C05469=1110.631,164.327,-63.571,-179.323,8.948,149.553
C05470=1110.636,164.078,-63.548,-179.324,8.945,149.553
C05471=1110.640,163.829,-63.525,-179.327,8.942,149.553
C05472=1110.644,163.580,-63.502,-179.329,8.939,149.553
C05473=1110.649,163.331,-63.479,-179.331,8.936,149.553
C05474=1110.654,163.082,-63.455,-179.334,8.932,149.552
C05475=1110.658,162.834,-63.432,-179.335,8.930,149.552
C05476=1110.663,162.585,-63.410,-179.338,8.926,149.552
C05477=1110.667,162.336,-63.387,-179.340,8.923,149.552
C05478=1110.672,162.087,-63.364,-179.342,8.920,149.552
C05479=1110.677,161.838,-63.341,-179.344,8.917,149.552
C05480=1110.681,161.588,-63.319,-179.346,8.914,149.551
C05481=1110.686,161.340,-63.296,-179.349,8.911,149.551
C05482=1110.690,161.091,-63.273,-179.351,8.907,149.551
C05483=1110.695,160.842,-63.249,-179.353,8.905,149.551
C05484=1110.699,160.593,-63.227,-179.355,8.902,149.551
C05485=1110.703,160.380,-63.208,-179.357,8.899,149.551
C05486=1110.707,160.167,-63.188,-179.359,8.896,149.551
C05487=1110.711,159.953,-63.168,-179.361,8.893,149.551
C05488=1110.715,159.739,-63.149,-179.362,8.891,149.550
C05489=1110.719,159.527,-63.129,-179.365,8.888,149.550
C05490=1110.723,159.312,-63.110,-179.366,8.885,149.550
C05491=1110.727,159.099,-63.090,-179.368,8.883,149.550
C05492=1110.731,158.886,-63.071,-179.369,8.880,149.550
C05493=1110.735,158.637,-63.048,-179.372,8.877,149.550
C05494=1110.740,158.388,-63.025,-179.374,8.873,149.550
C05495=1110.744,158.139,-63.003,-179.376,8.870,149.550
C05496=1110.750,157.890,-62.980,-179.379,8.867,149.549
C05497=1110.754,157.641,-62.958,-179.380,8.864,149.549
C05498=1110.758,157.392,-62.936,-179.382,8.861,149.549
C05499=1110.763,157.144,-62.913,-179.385,8.857,149.549
C05500=1110.767,156.895,-62.890,-179.387,8.854,149.549
C05501=1110.772,156.645,-62.867,-179.389,8.851,149.549
C05502=1110.777,156.397,-62.845,-179.391,8.847,149.548
C05503=1110.782,156.148,-62.822,-179.393,8.844,149.548
C05504=1110.786,155.899,-62.799,-179.395,8.841,149.548
C05505=1110.791,155.650,-62.778,-179.397,8.838,149.548
C05506=1110.795,155.401,-62.754,-179.399,8.834,149.548
C05507=1110.800,155.152,-62.732,-179.401,8.831,149.547
C05508=1110.805,154.903,-62.711,-179.404,8.828,149.547
C05509=1110.809,154.654,-62.687,-179.406,8.824,149.547
C05510=1110.814,154.405,-62.665,-179.408,8.821,149.547
C05511=1110.819,154.156,-62.642,-179.410,8.817,149.547
C05512=1110.823,153.907,-62.620,-179.412,8.815,149.546
C05513=1110.827,153.658,-62.598,-179.414,8.812,149.546
C05514=1110.833,153.409,-62.575,-179.416,8.808,149.546
C05515=1110.837,153.160,-62.553,-179.418,8.805,149.546
C05516=1110.841,152.911,-62.531,-179.420,8.801,149.546
C05517=1110.847,152.662,-62.508,-179.423,8.798,149.545
C05518=1110.851,152.413,-62.486,-179.425,8.794,149.545
C05519=1110.856,152.164,-62.464,-179.427,8.791,149.545
C05520=1110.860,151.916,-62.442,-179.429,8.788,149.545
C05521=1110.865,151.666,-62.419,-179.431,8.784,149.545
C05522=1110.870,151.417,-62.397,-179.433,8.781,149.544
C05523=1110.874,151.168,-62.375,-179.435,8.777,149.544
C05524=1110.878,150.920,-62.353,-179.438,8.774,149.544
C05525=1110.883,150.670,-62.330,-179.440,8.770,149.544
C05526=1110.888,150.422,-62.308,-179.442,8.767,149.543
C05527=1110.892,150.172,-62.286,-179.444,8.763,149.543
C05528=1110.897,149.924,-62.264,-179.446,8.760,149.543
C05529=1110.902,149.675,-62.241,-179.447,8.757,149.543
C05530=1110.906,149.425,-62.219,-179.449,8.753,149.543
C05531=1110.911,149.177,-62.198,-179.451,8.750,149.542
C05532=1110.915,148.927,-62.176,-179.454,8.747,149.542
C05533=1110.920,148.679,-62.154,-179.456,8.743,149.542
C05534=1110.925,148.429,-62.132,-179.458,8.740,149.542
C05535=1110.930,148.181,-62.109,-179.460,8.735,149.541
C05536=1110.934,147.932,-62.087,-179.463,8.732,149.541
C05537=1110.939,147.683,-62.065,-179.465,8.728,149.541
C05538=1110.943,147.434,-62.043,-179.466,8.724,149.540
C05539=1110.948,147.185,-62.021,-179.468,8.721,149.540
C05540=1110.952,146.936,-61.999,-179.470,8.717,149.540
C05541=1110.957,146.722,-61.981,-179.472,8.715,149.540
C05542=1110.960,146.508,-61.962,-179.474,8.711,149.539
C05543=1110.965,146.296,-61.943,-179.475,8.709,149.539
C05544=1110.968,146.082,-61.924,-179.477,8.705,149.539
C05545=1110.973,145.868,-61.905,-179.479,8.702,149.539
C05546=1110.977,145.654,-61.886,-179.481,8.699,149.539
C05547=1110.981,145.441,-61.868,-179.482,8.696,149.538
C05548=1110.985,145.227,-61.848,-179.485,8.693,149.538
C05549=1110.990,144.979,-61.827,-179.486,8.690,149.538
C05550=1110.994,144.730,-61.805,-179.488,8.686,149.537
C05551=1110.999,144.480,-61.784,-179.489,8.682,149.537
C05552=1111.004,144.232,-61.762,-179.491,8.679,149.537
C05553=1111.008,143.982,-61.740,-179.492,8.676,149.536
C05554=1111.013,143.734,-61.718,-179.494,8.672,149.536
C05555=1111.017,143.484,-61.696,-179.496,8.668,149.536
C05556=1111.022,143.236,-61.675,-179.497,8.666,149.535
C05557=1111.027,142.987,-61.653,-179.499,8.662,149.535
C05558=1111.031,142.738,-61.631,-179.501,8.658,149.535
C05559=1111.036,142.489,-61.609,-179.503,8.655,149.534
C05560=1111.041,142.239,-61.588,-179.504,8.652,149.534
C05561=1111.046,141.990,-61.566,-179.506,8.648,149.534
C05562=1111.049,141.741,-61.545,-179.507,8.645,149.533
C05563=1111.054,141.493,-61.523,-179.509,8.642,149.533
C05564=1111.059,141.244,-61.501,-179.511,8.638,149.533
C05565=1111.063,140.994,-61.480,-179.513,8.635,149.532
C05566=1111.068,140.745,-61.458,-179.515,8.631,149.532
C05567=1111.073,140.497,-61.437,-179.516,8.628,149.532
C05568=1111.077,140.247,-61.415,-179.518,8.624,149.532
C05569=1111.083,139.998,-61.394,-179.519,8.621,149.531
C05570=1111.087,139.750,-61.372,-179.521,8.618,149.531
C05571=1111.092,139.500,-61.350,-179.523,8.614,149.531
C05572=1111.097,139.251,-61.329,-179.524,8.611,149.530
C05573=1111.100,139.002,-61.307,-179.527,8.607,149.530
C05574=1111.105,138.753,-61.286,-179.529,8.604,149.530
C05575=1111.110,138.505,-61.264,-179.530,8.601,149.529
C05576=1111.115,138.255,-61.243,-179.532,8.597,149.529
C05577=1111.120,138.006,-61.221,-179.533,8.594,149.529
C05578=1111.125,137.757,-61.200,-179.535,8.591,149.528
C05579=1111.129,137.508,-61.179,-179.537,8.587,149.528
C05580=1111.133,137.259,-61.157,-179.538,8.583,149.528
C05581=1111.138,137.010,-61.136,-179.540,8.581,149.528
C05582=1111.143,136.761,-61.114,-179.542,8.577,149.527
C05583=1111.148,136.511,-61.093,-179.544,8.573,149.527
C05584=1111.152,136.263,-61.072,-179.545,8.571,149.527
C05585=1111.157,136.014,-61.050,-179.547,8.567,149.526
C05586=1111.161,135.764,-61.029,-179.549,8.563,149.526
C05587=1111.166,135.516,-61.007,-179.550,8.561,149.526
C05588=1111.171,135.267,-60.987,-179.552,8.557,149.525
C05589=1111.176,135.018,-60.965,-179.554,8.553,149.525
C05590=1111.180,134.768,-60.944,-179.555,8.550,149.525
C05591=1111.185,134.519,-60.922,-179.557,8.547,149.525
C05592=1111.189,134.271,-60.902,-179.560,8.544,149.524
C05593=1111.194,134.022,-60.880,-179.561,8.540,149.524
C05594=1111.199,133.772,-60.859,-179.563,8.537,149.524
C05595=1111.204,133.523,-60.837,-179.565,8.533,149.523
C05596=1111.208,133.274,-60.817,-179.566,8.530,149.523
C05597=1111.213,133.061,-60.798,-179.568,8.527,149.523
C05598=1111.217,132.846,-60.780,-179.569,8.524,149.523
C05599=1111.220,132.633,-60.762,-179.571,8.521,149.522
C05600=1111.224,132.420,-60.744,-179.572,8.519,149.522
C05601=1111.228,132.206,-60.726,-179.574,8.516,149.522
C05602=1111.233,131.992,-60.707,-179.575,8.513,149.522
C05603=1111.237,131.779,-60.689,-179.577,8.510,149.521
C05604=1111.241,131.565,-60.672,-179.578,8.507,149.521
C05605=1111.245,131.316,-60.650,-179.579,8.504,149.521
C05606=1111.250,131.067,-60.630,-179.582,8.500,149.521
C05607=1111.255,130.818,-60.609,-179.584,8.497,149.520
C05608=1111.260,130.569,-60.587,-179.585,8.494,149.520
C05609=1111.264,130.320,-60.567,-179.587,8.490,149.520
C05610=1111.269,130.071,-60.546,-179.589,8.487,149.519
C05611=1111.273,129.822,-60.524,-179.590,8.484,149.519
C05612=1111.278,129.572,-60.503,-179.592,8.481,149.519
C05613=1111.283,129.323,-60.482,-179.594,8.477,149.518
C05614=1111.288,129.074,-60.462,-179.595,8.474,149.518
C05615=1111.292,128.826,-60.440,-179.597,8.471,149.518
C05616=1111.297,128.577,-60.420,-179.599,8.467,149.518
C05617=1111.302,128.327,-60.399,-179.600,8.464,149.517
C05618=1111.306,128.078,-60.378,-179.603,8.461,149.517
C05619=1111.311,127.828,-60.357,-179.605,8.457,149.517
C05620=1111.315,127.580,-60.336,-179.606,8.454,149.517
C05621=1111.320,127.331,-60.315,-179.608,8.450,149.516
C05622=1111.326,127.082,-60.294,-179.610,8.447,149.516
C05623=1111.330,126.833,-60.274,-179.612,8.443,149.516
C05624=1111.335,126.583,-60.253,-179.613,8.441,149.516
C05625=1111.340,126.334,-60.232,-179.615,8.437,149.515
C05626=1111.345,126.086,-60.211,-179.617,8.433,149.515
C05627=1111.348,125.836,-60.190,-179.618,8.431,149.515
C05628=1111.353,125.587,-60.170,-179.620,8.427,149.514
C05629=1111.358,125.338,-60.149,-179.622,8.423,149.514
C05630=1111.362,125.089,-60.128,-179.624,8.421,149.514
C05631=1111.368,124.840,-60.107,-179.626,8.417,149.514
C05632=1111.372,124.591,-60.087,-179.628,8.414,149.513
C05633=1111.377,124.342,-60.066,-179.629,8.410,149.513
C05634=1111.382,124.093,-60.046,-179.631,8.407,149.513
C05635=1111.386,123.844,-60.025,-179.633,8.403,149.512
C05636=1111.391,123.594,-60.004,-179.634,8.401,149.512
C05637=1111.396,123.345,-59.984,-179.636,8.397,149.512
C05638=1111.401,123.096,-59.963,-179.638,8.393,149.512
C05639=1111.405,122.847,-59.942,-179.639,8.391,149.511
C05640=1111.410,122.598,-59.922,-179.641,8.387,149.511
C05641=1111.415,122.349,-59.901,-179.643,8.384,149.511
C05642=1111.419,122.100,-59.881,-179.645,8.380,149.510
C05643=1111.424,121.851,-59.860,-179.647,8.377,149.510
C05644=1111.429,121.602,-59.839,-179.649,8.374,149.510
C05645=1111.433,121.353,-59.819,-179.651,8.370,149.510
C05646=1111.439,121.104,-59.798,-179.652,8.367,149.509
C05647=1111.443,120.855,-59.778,-179.654,8.363,149.509
C05648=1111.448,120.605,-59.758,-179.656,8.360,149.509
C05649=1111.452,120.356,-59.738,-179.657,8.357,149.509
C05650=1111.457,120.107,-59.717,-179.659,8.353,149.508
C05651=1111.462,119.858,-59.696,-179.661,8.350,149.508
C05652=1111.466,119.609,-59.676,-179.663,8.346,149.508
C05653=1111.470,119.395,-59.659,-179.664,8.344,149.507
C05654=1111.475,119.181,-59.641,-179.666,8.341,149.507
C05655=1111.478,118.967,-59.623,-179.667,8.338,149.507
C05656=1111.483,118.753,-59.606,-179.668,8.335,149.507
C05657=1111.487,118.540,-59.588,-179.670,8.332,149.506
C05658=1111.491,118.326,-59.570,-179.672,8.329,149.506
C05659=1111.494,118.113,-59.554,-179.673,8.326,149.506
C05660=1111.499,117.899,-59.536,-179.675,8.323,149.506
C05661=1111.504,117.650,-59.515,-179.677,8.320,149.505
C05662=1111.509,117.400,-59.496,-179.679,8.316,149.505
C05663=1111.513,117.151,-59.475,-179.680,8.313,149.505
C05664=1111.517,116.902,-59.455,-179.682,8.310,149.505
C05665=1111.522,116.653,-59.435,-179.684,8.306,149.504
C05666=1111.527,116.403,-59.414,-179.685,8.303,149.504
C05667=1111.532,116.155,-59.394,-179.687,8.300,149.504
C05668=1111.537,115.906,-59.375,-179.689,8.296,149.503
C05669=1111.542,115.657,-59.354,-179.691,8.293,149.503
C05670=1111.546,115.408,-59.334,-179.692,8.290,149.503
C05671=1111.551,115.158,-59.314,-179.694,8.286,149.503
C05672=1111.556,114.909,-59.293,-179.696,8.283,149.502
C05673=1111.560,114.660,-59.273,-179.698,8.279,149.502
C05674=1111.565,114.410,-59.253,-179.699,8.276,149.502
C05675=1111.570,114.162,-59.233,-179.701,8.273,149.501
C05676=1111.575,113.913,-59.213,-179.703,8.269,149.501
C05677=1111.579,113.664,-59.193,-179.705,8.265,149.501
C05678=1111.584,113.415,-59.173,-179.706,8.262,149.501
C05679=1111.589,113.165,-59.152,-179.708,8.259,149.500
C05680=1111.594,112.916,-59.132,-179.710,8.255,149.500
C05681=1111.599,112.667,-59.113,-179.712,8.252,149.500
C05682=1111.603,112.418,-59.092,-179.713,8.249,149.499
C05683=1111.608,112.168,-59.073,-179.715,8.245,149.499
C05684=1111.613,111.919,-59.052,-179.717,8.242,149.499
C05685=1111.617,111.670,-59.033,-179.719,8.238,149.498
C05686=1111.622,111.421,-59.012,-179.720,8.235,149.498
C05687=1111.627,111.172,-58.993,-179.722,8.231,149.498
C05688=1111.632,110.923,-58.973,-179.724,8.228,149.497
C05689=1111.636,110.674,-58.953,-179.726,8.224,149.497
C05690=1111.641,110.424,-58.933,-179.728,8.221,149.497
C05691=1111.646,110.176,-58.913,-179.730,8.217,149.497
C05692=1111.651,109.926,-58.894,-179.733,8.213,149.497
C05693=1111.656,109.677,-58.874,-179.734,8.209,149.496
C05694=1111.660,109.428,-58.854,-179.736,8.205,149.496
C05695=1111.665,109.178,-58.834,-179.739,8.202,149.496
C05696=1111.670,108.930,-58.814,-179.740,8.198,149.495
C05697=1111.675,108.680,-58.794,-179.742,8.194,149.495
C05698=1111.679,108.431,-58.775,-179.744,8.191,149.495
C05699=1111.684,108.182,-58.754,-179.746,8.187,149.494
C05700=1111.689,107.933,-58.735,-179.748,8.184,149.494
C05701=1111.694,107.683,-58.715,-179.750,8.180,149.494
C05702=1111.699,107.434,-58.696,-179.752,8.176,149.493
C05703=1111.704,107.186,-58.676,-179.754,8.173,149.493
C05704=1111.708,106.936,-58.656,-179.755,8.169,149.493
C05705=1111.713,106.686,-58.636,-179.757,8.165,149.493
C05706=1111.717,106.437,-58.617,-179.759,8.162,149.492
C05707=1111.722,106.189,-58.597,-179.761,8.158,149.492
C05708=1111.727,105.939,-58.578,-179.763,8.154,149.492
C05709=1111.731,105.725,-58.561,-179.765,8.151,149.491
C05710=1111.735,105.511,-58.544,-179.766,8.148,149.491
C05711=1111.739,105.298,-58.527,-179.768,8.144,149.491
C05712=1111.743,105.084,-58.511,-179.769,8.141,149.490
C05713=1111.748,104.870,-58.494,-179.771,8.138,149.490
C05714=1111.752,104.656,-58.478,-179.773,8.135,149.490
C05715=1111.756,104.443,-58.460,-179.774,8.131,149.490
C05716=1111.760,104.228,-58.444,-179.776,8.128,149.489
C05717=1111.764,103.979,-58.424,-179.777,8.124,149.489
C05718=1111.770,103.730,-58.405,-179.779,8.121,149.489
C05719=1111.774,103.481,-58.385,-179.781,8.117,149.488
C05720=1111.778,103.232,-58.366,-179.783,8.114,149.488
C05721=1111.784,102.983,-58.346,-179.785,8.110,149.488
C05722=1111.788,102.733,-58.327,-179.786,8.106,149.487
C05723=1111.793,102.484,-58.307,-179.788,8.102,149.487
C05724=1111.798,102.235,-58.288,-179.790,8.098,149.486
C05725=1111.802,101.986,-58.269,-179.791,8.095,149.486
C05726=1111.808,101.737,-58.249,-179.793,8.091,149.486
C05727=1111.813,101.487,-58.230,-179.795,8.087,149.485
C05728=1111.817,101.238,-58.211,-179.797,8.083,149.485
C05729=1111.822,100.989,-58.191,-179.798,8.079,149.484
C05730=1111.827,100.740,-58.172,-179.800,8.075,149.484
C05731=1111.832,100.491,-58.152,-179.801,8.072,149.484
C05732=1111.836,100.241,-58.133,-179.804,8.068,149.483
C05733=1111.841,99.993,-58.114,-179.805,8.064,149.483
C05734=1111.846,99.742,-58.095,-179.807,8.060,149.483
C05735=1111.850,99.493,-58.076,-179.808,8.056,149.482
C05736=1111.856,99.244,-58.057,-179.810,8.053,149.482
C05737=1111.860,98.995,-58.037,-179.812,8.049,149.481
C05738=1111.865,98.746,-58.018,-179.813,8.046,149.481
C05739=1111.870,98.497,-57.999,-179.815,8.042,149.481
C05740=1111.874,98.248,-57.980,-179.816,8.038,149.480
C05741=1111.879,97.998,-57.960,-179.818,8.034,149.480
C05742=1111.885,97.749,-57.942,-179.819,8.030,149.479
C05743=1111.889,97.500,-57.923,-179.821,8.027,149.479
C05744=1111.894,97.251,-57.904,-179.823,8.023,149.478
C05745=1111.898,97.002,-57.885,-179.824,8.019,149.478
C05746=1111.903,96.753,-57.865,-179.826,8.015,149.478
C05747=1111.909,96.503,-57.846,-179.827,8.011,149.477
C05748=1111.913,96.254,-57.828,-179.829,8.007,149.477
C05749=1111.918,96.004,-57.808,-179.830,8.004,149.476
C05750=1111.922,95.756,-57.789,-179.832,8.000,149.476
C05751=1111.928,95.506,-57.770,-179.833,7.996,149.475
C05752=1111.932,95.257,-57.752,-179.835,7.992,149.475
C05753=1111.937,95.008,-57.732,-179.836,7.988,149.474
C05754=1111.942,94.758,-57.714,-179.838,7.985,149.474
C05755=1111.947,94.509,-57.694,-179.840,7.981,149.474
C05756=1111.951,94.260,-57.676,-179.841,7.978,149.473
C05757=1111.956,94.010,-57.657,-179.842,7.973,149.473
C05758=1111.961,93.762,-57.638,-179.843,7.969,149.472
C05759=1111.966,93.513,-57.619,-179.845,7.965,149.472
C05760=1111.970,93.263,-57.600,-179.846,7.962,149.471
C05761=1111.976,93.014,-57.581,-179.848,7.958,149.471
C05762=1111.980,92.764,-57.563,-179.849,7.955,149.470
C05763=1111.985,92.515,-57.543,-179.851,7.951,149.470
C05764=1111.989,92.266,-57.524,-179.852,7.946,149.469
C05765=1111.994,92.053,-57.509,-179.853,7.944,149.469
C05766=1111.998,91.838,-57.492,-179.855,7.940,149.469
C05767=1112.002,91.624,-57.476,-179.856,7.937,149.468
C05768=1112.007,91.411,-57.460,-179.857,7.934,149.468
C05769=1112.011,91.197,-57.444,-179.858,7.930,149.467
C05770=1112.014,90.982,-57.428,-179.859,7.927,149.467
C05771=1112.019,90.769,-57.412,-179.860,7.923,149.466
C05772=1112.023,90.555,-57.395,-179.861,7.920,149.466
C05773=1112.028,90.305,-57.377,-179.863,7.916,149.466
C05774=1112.032,90.056,-57.358,-179.864,7.913,149.465
C05775=1112.038,89.807,-57.340,-179.865,7.909,149.465
C05776=1112.042,89.557,-57.321,-179.867,7.905,149.464
C05777=1112.048,89.308,-57.302,-179.868,7.901,149.464
C05778=1112.052,89.059,-57.284,-179.870,7.897,149.463
C05779=1112.056,88.810,-57.265,-179.870,7.894,149.463
C05780=1112.062,88.560,-57.247,-179.872,7.890,149.462
C05781=1112.067,88.311,-57.228,-179.873,7.886,149.462
C05782=1112.071,88.062,-57.210,-179.875,7.882,149.461
C05783=1112.076,87.813,-57.190,-179.876,7.879,149.461
C05784=1112.081,87.564,-57.172,-179.877,7.875,149.460
C05785=1112.086,87.314,-57.154,-179.878,7.871,149.460
C05786=1112.090,87.065,-57.135,-179.879,7.867,149.459
C05787=1112.096,86.816,-57.117,-179.881,7.864,149.459
C05788=1112.100,86.566,-57.098,-179.882,7.859,149.458
C05789=1112.105,86.317,-57.080,-179.883,7.856,149.458
C05790=1112.110,86.068,-57.061,-179.884,7.852,149.457
C05791=1112.115,85.818,-57.043,-179.886,7.848,149.457
C05792=1112.119,85.569,-57.024,-179.887,7.845,149.456
C05793=1112.124,85.320,-57.006,-179.888,7.841,149.455
C05794=1112.130,85.071,-56.987,-179.889,7.837,149.455
C05795=1112.134,84.821,-56.968,-179.890,7.833,149.454
C05796=1112.139,84.572,-56.950,-179.891,7.829,149.454
C05797=1112.144,84.323,-56.932,-179.893,7.825,149.454
C05798=1112.148,84.073,-56.914,-179.894,7.822,149.453
C05799=1112.153,83.824,-56.895,-179.895,7.818,149.452
C05800=1112.158,83.575,-56.877,-179.896,7.814,149.452
C05801=1112.163,83.326,-56.859,-179.897,7.811,149.451
C05802=1112.167,83.076,-56.840,-179.898,7.806,149.451
C05803=1112.172,82.827,-56.823,-179.899,7.803,149.450
C05804=1112.178,82.578,-56.803,-179.900,7.799,149.450
C05805=1112.183,82.329,-56.785,-179.902,7.795,149.449
C05806=1112.188,82.080,-56.767,-179.903,7.792,149.449
C05807=1112.192,81.830,-56.749,-179.904,7.788,149.448
C05808=1112.197,81.581,-56.731,-179.905,7.784,149.447
C05809=1112.202,81.331,-56.713,-179.906,7.780,149.447
C05810=1112.207,81.083,-56.694,-179.907,7.777,149.446
C05811=1112.211,80.833,-56.675,-179.908,7.773,149.446
C05812=1112.216,80.583,-56.657,-179.909,7.769,149.445
C05813=1112.221,80.334,-56.639,-179.910,7.766,149.445
C05814=1112.226,80.085,-56.621,-179.911,7.762,149.444
C05815=1112.231,79.836,-56.603,-179.912,7.758,149.444
C05816=1112.235,79.586,-56.585,-179.914,7.754,149.443
C05817=1112.240,79.337,-56.567,-179.915,7.751,149.443
C05818=1112.245,79.088,-56.549,-179.916,7.746,149.442
C05819=1112.250,78.839,-56.531,-179.917,7.743,149.442
C05820=1112.256,78.589,-56.513,-179.917,7.740,149.441
C05821=1112.259,78.375,-56.497,-179.918,7.737,149.441
C05822=1112.264,78.161,-56.482,-179.919,7.734,149.440
C05823=1112.267,77.947,-56.466,-179.920,7.730,149.439
C05824=1112.272,77.733,-56.451,-179.921,7.727,149.439
C05825=1112.276,77.519,-56.435,-179.922,7.724,149.439
C05826=1112.281,77.305,-56.420,-179.922,7.721,149.438
C05827=1112.284,77.091,-56.404,-179.923,7.718,149.438
C05828=1112.289,76.877,-56.389,-179.924,7.714,149.437
C05829=1112.293,76.627,-56.370,-179.925,7.710,149.437
C05830=1112.298,76.378,-56.352,-179.927,7.706,149.436
C05831=1112.303,76.129,-56.334,-179.929,7.702,149.436
C05832=1112.308,75.880,-56.316,-179.930,7.698,149.435
C05833=1112.313,75.630,-56.298,-179.931,7.694,149.435
C05834=1112.318,75.381,-56.280,-179.933,7.690,149.434
C05835=1112.323,75.132,-56.262,-179.934,7.686,149.434
C05836=1112.328,74.883,-56.244,-179.936,7.682,149.433
C05837=1112.332,74.633,-56.226,-179.937,7.678,149.433
C05838=1112.337,74.383,-56.209,-179.939,7.674,149.432
C05839=1112.342,74.134,-56.191,-179.939,7.671,149.432
C05840=1112.346,73.885,-56.173,-179.941,7.667,149.431
C05841=1112.351,73.636,-56.155,-179.942,7.663,149.431
C05842=1112.356,73.387,-56.138,-179.944,7.659,149.430
C05843=1112.361,73.138,-56.120,-179.945,7.655,149.430
C05844=1112.366,72.888,-56.102,-179.947,7.651,149.429
C05845=1112.371,72.639,-56.084,-179.948,7.647,149.429
C05846=1112.376,72.389,-56.066,-179.949,7.643,149.428
C05847=1112.381,72.140,-56.048,-179.951,7.639,149.428
C05848=1112.386,71.891,-56.030,-179.953,7.635,149.427
C05849=1112.391,71.642,-56.014,-179.954,7.631,149.427
C05850=1112.395,71.392,-55.996,-179.955,7.628,149.426
C05851=1112.400,71.143,-55.978,-179.956,7.624,149.426
C05852=1112.406,70.893,-55.960,-179.957,7.619,149.425
C05853=1112.410,70.644,-55.942,-179.959,7.616,149.425
C05854=1112.415,70.395,-55.924,-179.960,7.612,149.424
C05855=1112.420,70.146,-55.908,-179.962,7.607,149.424
C05856=1112.425,69.896,-55.890,-179.963,7.603,149.423
C05857=1112.430,69.647,-55.872,-179.965,7.600,149.423
C05858=1112.435,69.397,-55.855,-179.966,7.596,149.422
C05859=1112.440,69.148,-55.837,-179.967,7.591,149.422
C05860=1112.445,68.899,-55.819,-179.968,7.588,149.421
C05861=1112.449,68.650,-55.802,-179.969,7.584,149.421
C05862=1112.454,68.400,-55.784,-179.971,7.580,149.420
C05863=1112.459,68.151,-55.766,-179.973,7.576,149.420
C05864=1112.464,67.901,-55.749,-179.974,7.572,149.419
C05865=1112.468,67.653,-55.731,-179.975,7.568,149.419
C05866=1112.474,67.403,-55.714,-179.977,7.564,149.418
C05867=1112.479,67.154,-55.696,-179.978,7.560,149.418
C05868=1112.484,66.904,-55.679,-179.980,7.556,149.417
C05869=1112.488,66.655,-55.661,-179.980,7.553,149.417
C05870=1112.493,66.405,-55.644,-179.982,7.548,149.416
C05871=1112.498,66.156,-55.626,-179.983,7.545,149.416
C05872=1112.503,65.907,-55.610,-179.985,7.541,149.415
C05873=1112.507,65.657,-55.592,-179.986,7.536,149.415
C05874=1112.513,65.408,-55.574,-179.987,7.532,149.414
C05875=1112.517,65.159,-55.557,-179.988,7.528,149.413
C05876=1112.522,64.909,-55.540,-179.990,7.524,149.413
C05877=1112.527,64.695,-55.525,-179.991,7.521,149.413
C05878=1112.531,64.481,-55.510,-179.992,7.518,149.412
C05879=1112.535,64.266,-55.495,-179.994,7.514,149.412
C05880=1112.539,64.053,-55.480,-179.994,7.511,149.411
C05881=1112.544,63.839,-55.465,-179.995,7.508,149.411
C05882=1112.547,63.624,-55.451,-179.996,7.505,149.410
C05883=1112.552,63.410,-55.436,-179.998,7.501,149.410
C05884=1112.556,63.197,-55.421,-179.999,7.498,149.410
C05885=1112.561,62.947,-55.403,-180.000,7.493,149.409
C05886=1112.566,62.698,-55.386,179.998,7.490,149.409
C05887=1112.570,62.448,-55.369,179.997,7.485,149.408
C05888=1112.575,62.199,-55.351,179.996,7.481,149.407
C05889=1112.580,61.950,-55.335,179.995,7.478,149.407
C05890=1112.586,61.700,-55.318,179.994,7.474,149.406
C05891=1112.590,61.451,-55.300,179.992,7.470,149.406
C05892=1112.595,61.202,-55.283,179.991,7.466,149.405
C05893=1112.600,60.952,-55.266,179.990,7.462,149.405
C05894=1112.605,60.702,-55.249,179.988,7.458,149.404
C05895=1112.610,60.453,-55.231,179.987,7.454,149.404
C05896=1112.615,60.205,-55.215,179.986,7.450,149.403
C05897=1112.620,59.955,-55.198,179.985,7.446,149.403
C05898=1112.624,59.705,-55.181,179.984,7.442,149.402
C05899=1112.629,59.456,-55.163,179.982,7.438,149.402
C05900=1112.634,59.207,-55.146,179.981,7.434,149.401
C05901=1112.639,58.957,-55.129,179.980,7.430,149.400
C05902=1112.644,58.708,-55.113,179.978,7.426,149.400
C05903=1112.649,58.458,-55.095,179.977,7.422,149.399
C05904=1112.653,58.209,-55.078,179.976,7.418,149.399
C05905=1112.659,57.960,-55.061,179.975,7.414,149.398
C05906=1112.664,57.711,-55.044,179.973,7.410,149.398
C05907=1112.669,57.461,-55.027,179.972,7.406,149.397
C05908=1112.673,57.211,-55.011,179.971,7.402,149.397
C05909=1112.679,56.962,-54.993,179.970,7.399,149.396
C05910=1112.684,56.713,-54.977,179.969,7.395,149.396
C05911=1112.689,56.463,-54.960,179.967,7.390,149.395
C05912=1112.693,56.214,-54.942,179.966,7.386,149.395
C05913=1112.698,55.965,-54.926,179.965,7.382,149.394
C05914=1112.703,55.716,-54.909,179.964,7.378,149.393
C05915=1112.708,55.466,-54.892,179.962,7.374,149.393
C05916=1112.713,55.216,-54.875,179.962,7.370,149.392
C05917=1112.718,54.967,-54.858,179.960,7.367,149.392
C05918=1112.723,54.718,-54.842,179.959,7.362,149.391
C05919=1112.728,54.468,-54.825,179.957,7.358,149.391
C05920=1112.732,54.219,-54.808,179.956,7.354,149.390
C05921=1112.737,53.970,-54.792,179.955,7.350,149.390
C05922=1112.743,53.720,-54.774,179.954,7.347,149.389
C05923=1112.747,53.471,-54.758,179.953,7.343,149.389
C05924=1112.752,53.222,-54.741,179.952,7.338,149.388
C05925=1112.757,52.972,-54.724,179.951,7.334,149.387
C05926=1112.762,52.723,-54.707,179.949,7.330,149.387
C05927=1112.767,52.474,-54.691,179.948,7.326,149.386
C05928=1112.772,52.224,-54.674,179.947,7.323,149.386
C05929=1112.777,51.974,-54.658,179.946,7.318,149.385
C05930=1112.782,51.725,-54.642,179.945,7.314,149.384
C05931=1112.787,51.475,-54.624,179.943,7.310,149.384
C05932=1112.792,51.226,-54.608,179.942,7.306,149.383
C05933=1112.796,51.012,-54.593,179.941,7.303,149.383
C05934=1112.800,50.798,-54.580,179.940,7.300,149.383
C05935=1112.805,50.584,-54.565,179.939,7.295,149.382
C05936=1112.809,50.370,-54.551,179.938,7.292,149.381
C05937=1112.813,50.155,-54.537,179.937,7.289,149.381
C05938=1112.817,49.941,-54.522,179.936,7.286,149.381
C05939=1112.822,49.726,-54.508,179.935,7.282,149.380
C05940=1112.826,49.513,-54.494,179.934,7.279,149.379
C05941=1112.831,49.264,-54.477,179.933,7.274,149.379
C05942=1112.836,49.014,-54.461,179.932,7.270,149.378
C05943=1112.840,48.764,-54.445,179.931,7.267,149.378
C05944=1112.846,48.515,-54.428,179.930,7.263,149.377
C05945=1112.850,48.266,-54.411,179.929,7.259,149.377
C05946=1112.856,48.016,-54.396,179.928,7.254,149.376
C05947=1112.860,47.767,-54.379,179.927,7.250,149.375
C05948=1112.865,47.517,-54.362,179.925,7.246,149.375
C05949=1112.870,47.268,-54.346,179.925,7.243,149.374
C05950=1112.875,47.018,-54.329,179.923,7.238,149.374
C05951=1112.881,46.769,-54.313,179.922,7.234,149.373
C05952=1112.885,46.520,-54.296,179.921,7.230,149.373
C05953=1112.890,46.270,-54.280,179.920,7.226,149.372
C05954=1112.895,46.021,-54.264,179.919,7.221,149.371
C05955=1112.899,45.771,-54.247,179.918,7.218,149.371
C05956=1112.905,45.522,-54.232,179.917,7.214,149.370
C05957=1112.910,45.272,-54.215,179.916,7.210,149.369
C05958=1112.915,45.023,-54.198,179.915,7.205,149.369
C05959=1112.920,44.773,-54.182,179.913,7.202,149.368
C05960=1112.925,44.525,-54.166,179.913,7.198,149.368
C05961=1112.929,44.275,-54.149,179.911,7.194,149.367
C05962=1112.935,44.026,-54.134,179.910,7.189,149.366
C05963=1112.939,43.776,-54.117,179.909,7.185,149.366
C05964=1112.945,43.527,-54.102,179.908,7.181,149.365
C05965=1112.949,43.277,-54.085,179.907,7.177,149.365
C05966=1112.954,43.028,-54.069,179.906,7.173,149.364
C05967=1112.959,42.778,-54.053,179.905,7.169,149.364
C05968=1112.964,42.529,-54.037,179.904,7.165,149.363
C05969=1112.969,42.279,-54.020,179.902,7.161,149.362
C05970=1112.974,42.030,-54.005,179.901,7.157,149.362
C05971=1112.979,41.781,-53.988,179.901,7.153,149.361
C05972=1112.984,41.531,-53.972,179.900,7.149,149.360
C05973=1112.989,41.282,-53.956,179.898,7.145,149.360
C05974=1112.994,41.032,-53.940,179.897,7.141,149.359
C05975=1112.998,40.783,-53.924,179.896,7.136,149.359
C05976=1113.004,40.533,-53.908,179.895,7.132,149.358
C05977=1113.009,40.285,-53.892,179.895,7.128,149.357
C05978=1113.014,40.035,-53.876,179.894,7.124,149.357
C05979=1113.019,39.786,-53.859,179.893,7.120,149.356
C05980=1113.024,39.536,-53.843,179.891,7.116,149.356
C05981=1113.029,39.286,-53.828,179.890,7.112,149.355
C05982=1113.033,39.037,-53.811,179.889,7.108,149.354
C05983=1113.039,38.787,-53.796,179.888,7.104,149.354
C05984=1113.044,38.538,-53.780,179.887,7.099,149.353
C05985=1113.049,38.288,-53.763,179.886,7.095,149.352
C05986=1113.054,38.039,-53.748,179.885,7.091,149.352
C05987=1113.059,37.789,-53.732,179.884,7.087,149.351
C05988=1113.064,37.540,-53.716,179.884,7.083,149.350
C05989=1113.067,37.326,-53.702,179.882,7.079,149.350
C05990=1113.072,37.112,-53.689,179.882,7.076,149.349
C05991=1113.076,36.898,-53.675,179.881,7.072,149.349
C05992=1113.080,36.683,-53.661,179.880,7.068,149.348
C05993=1113.085,36.469,-53.648,179.879,7.065,149.348
C05994=1113.089,36.255,-53.634,179.878,7.061,149.347
C05995=1113.093,36.040,-53.620,179.877,7.058,149.347
C05996=1113.098,35.825,-53.607,179.876,7.054,149.346
C05997=1113.103,35.576,-53.591,179.876,7.050,149.345
C05998=1113.108,35.327,-53.575,179.875,7.046,149.345
C05999=1113.112,35.077,-53.560,179.874,7.042,149.344
C06000=1113.118,34.828,-53.544,179.873,7.038,149.343
C06001=1113.123,34.579,-53.528,179.872,7.033,149.343
C06002=1113.128,34.329,-53.512,179.871,7.029,149.342
C06003=1113.133,34.080,-53.496,179.870,7.025,149.341
C06004=1113.138,33.830,-53.481,179.869,7.021,149.341
C06005=1113.142,33.580,-53.466,179.868,7.017,149.340
C06006=1113.148,33.332,-53.449,179.867,7.013,149.339
C06007=1113.153,33.082,-53.434,179.866,7.008,149.339
C06008=1113.158,32.832,-53.418,179.865,7.004,149.338
C06009=1113.162,32.583,-53.403,179.864,7.000,149.338
C06010=1113.168,32.334,-53.387,179.863,6.996,149.337
C06011=1113.173,32.084,-53.371,179.862,6.992,149.336
C06012=1113.178,31.834,-53.356,179.861,6.987,149.336
C06013=1113.183,31.585,-53.341,179.861,6.983,149.335
C06014=1113.188,31.336,-53.325,179.860,6.979,149.334
C06015=1113.193,31.086,-53.309,179.859,6.975,149.333
C06016=1113.198,30.837,-53.293,179.858,6.971,149.333
C06017=1113.202,30.588,-53.278,179.857,6.966,149.332
C06018=1113.208,30.338,-53.262,179.856,6.962,149.331
C06019=1113.213,30.088,-53.246,179.855,6.958,149.331
C06020=1113.217,29.839,-53.231,179.854,6.954,149.330
C06021=1113.223,29.590,-53.216,179.854,6.949,149.329
C06022=1113.228,29.340,-53.200,179.853,6.945,149.329
C06023=1113.232,29.090,-53.185,179.852,6.941,149.328
C06024=1113.237,28.841,-53.169,179.851,6.937,149.327
C06025=1113.243,28.592,-53.153,179.850,6.932,149.327
C06026=1113.248,28.343,-53.138,179.849,6.929,149.326
C06027=1113.252,28.092,-53.123,179.849,6.924,149.325
C06028=1113.257,27.843,-53.108,179.848,6.920,149.324
C06029=1113.263,27.593,-53.093,179.846,6.915,149.324
C06030=1113.268,27.344,-53.077,179.845,6.911,149.323
C06031=1113.273,27.095,-53.062,179.844,6.907,149.322
C06032=1113.277,26.845,-53.046,179.844,6.903,149.322
C06033=1113.283,26.595,-53.031,179.843,6.899,149.321
C06034=1113.288,26.346,-53.016,179.842,6.894,149.320
C06035=1113.293,26.097,-53.000,179.841,6.890,149.320
C06036=1113.298,25.848,-52.985,179.841,6.885,149.319
C06037=1113.302,25.598,-52.969,179.840,6.881,149.318
C06038=1113.307,25.348,-52.955,179.839,6.877,149.317
C06039=1113.313,25.099,-52.939,179.838,6.873,149.317
C06040=1113.318,24.849,-52.924,179.838,6.868,149.316
C06041=1113.323,24.600,-52.909,179.836,6.864,149.315
C06042=1113.328,24.351,-52.893,179.835,6.860,149.315
C06043=1113.332,24.100,-52.878,179.835,6.855,149.314
C06044=1113.338,23.851,-52.863,179.834,6.851,149.313
C06045=1113.342,23.638,-52.850,179.833,6.847,149.312
C06046=1113.347,23.423,-52.837,179.833,6.844,149.312
C06047=1113.351,23.208,-52.823,179.833,6.840,149.311
C06048=1113.355,22.994,-52.811,179.831,6.836,149.311
C06049=1113.359,22.779,-52.797,179.831,6.833,149.310
C06050=1113.364,22.565,-52.785,179.830,6.829,149.309
C06051=1113.368,22.351,-52.771,179.829,6.825,149.309
C06052=1113.372,22.136,-52.758,179.829,6.821,149.308
C06053=1113.377,21.887,-52.743,179.828,6.817,149.307
C06054=1113.383,21.637,-52.729,179.827,6.812,149.306
C06055=1113.387,21.388,-52.714,179.827,6.809,149.306
C06056=1113.392,21.139,-52.699,179.826,6.804,149.305
C06057=1113.397,20.888,-52.683,179.825,6.800,149.304
C06058=1113.402,20.639,-52.668,179.824,6.795,149.303
C06059=1113.407,20.390,-52.653,179.823,6.791,149.303
C06060=1113.412,20.140,-52.639,179.822,6.786,149.302
C06061=1113.418,19.890,-52.623,179.822,6.782,149.301
C06062=1113.422,19.641,-52.608,179.821,6.778,149.301
C06063=1113.427,19.392,-52.594,179.821,6.773,149.300
C06064=1113.433,19.142,-52.578,179.820,6.769,149.299
C06065=1113.437,18.893,-52.563,179.819,6.764,149.298
C06066=1113.443,18.643,-52.548,179.818,6.760,149.297
C06067=1113.447,18.394,-52.533,179.818,6.755,149.297
C06068=1113.452,18.144,-52.519,179.817,6.751,149.296
C06069=1113.458,17.895,-52.503,179.817,6.747,149.295
C06070=1113.463,17.645,-52.489,179.816,6.743,149.294
C06071=1113.467,17.396,-52.474,179.815,6.738,149.294
C06072=1113.473,17.146,-52.459,179.814,6.734,149.293
C06073=1113.478,16.897,-52.444,179.813,6.729,149.292
C06074=1113.483,16.647,-52.430,179.813,6.724,149.291
C06075=1113.488,16.398,-52.414,179.812,6.720,149.290
C06076=1113.493,16.148,-52.400,179.811,6.715,149.290
C06077=1113.498,15.899,-52.385,179.811,6.712,149.289
C06078=1113.503,15.649,-52.370,179.810,6.707,149.288
C06079=1113.508,15.400,-52.355,179.810,6.702,149.287
C06080=1113.513,15.150,-52.341,179.809,6.698,149.286
C06081=1113.518,14.901,-52.326,179.808,6.693,149.286
C06082=1113.523,14.651,-52.311,179.807,6.689,149.285
C06083=1113.528,14.402,-52.296,179.806,6.684,149.284
C06084=1113.533,14.152,-52.282,179.806,6.680,149.283
C06085=1113.538,13.903,-52.268,179.806,6.676,149.283
C06086=1113.543,13.653,-52.252,179.805,6.671,149.282
C06087=1113.548,13.404,-52.238,179.804,6.667,149.281
C06088=1113.553,13.154,-52.223,179.803,6.662,149.280
C06089=1113.558,12.905,-52.208,179.803,6.658,149.279
C06090=1113.564,12.655,-52.194,179.802,6.653,149.278
C06091=1113.568,12.406,-52.179,179.802,6.648,149.277
C06092=1113.573,12.156,-52.164,179.801,6.644,149.277
C06093=1113.578,11.906,-52.150,179.800,6.639,149.276
C06094=1113.583,11.657,-52.135,179.800,6.635,149.275
C06095=1113.588,11.407,-52.120,179.800,6.631,149.274
C06096=1113.593,11.157,-52.106,179.799,6.626,149.273
C06097=1113.598,10.908,-52.091,179.798,6.622,149.273
C06098=1113.604,10.659,-52.077,179.798,6.617,149.272
C06099=1113.609,10.410,-52.063,179.797,6.612,149.271
C06100=1113.614,10.160,-52.048,179.796,6.608,149.270
C06101=1113.618,9.945,-52.035,179.796,6.604,149.269
C06102=1113.622,9.730,-52.023,179.795,6.600,149.269
C06103=1113.627,9.516,-52.010,179.795,6.596,149.268
C06104=1113.631,9.301,-51.998,179.795,6.592,149.267
C06105=1113.636,9.087,-51.986,179.794,6.588,149.266
C06106=1113.640,8.873,-51.973,179.793,6.584,149.266
C06107=1113.644,8.658,-51.961,179.793,6.580,149.265
C06108=1113.648,8.444,-51.949,179.792,6.576,149.264
C06109=1113.653,8.194,-51.934,179.792,6.571,149.263
C06110=1113.658,7.945,-51.919,179.791,6.567,149.262
C06111=1113.663,7.695,-51.905,179.791,6.563,149.262
C06112=1113.669,7.445,-51.890,179.790,6.558,149.261
C06113=1113.674,7.196,-51.876,179.790,6.554,149.260
C06114=1113.679,6.947,-51.862,179.789,6.549,149.259
C06115=1113.684,6.697,-51.848,179.789,6.544,149.258
C06116=1113.689,6.447,-51.833,179.788,6.540,149.257
C06117=1113.694,6.198,-51.818,179.787,6.535,149.257
C06118=1113.699,5.948,-51.804,179.786,6.531,149.256
C06119=1113.704,5.699,-51.790,179.786,6.526,149.255
C06120=1113.709,5.450,-51.776,179.785,6.521,149.254
C06121=1113.714,5.200,-51.762,179.785,6.516,149.253
C06122=1113.719,4.950,-51.747,179.784,6.513,149.252
C06123=1113.724,4.701,-51.733,179.784,6.508,149.252
C06124=1113.729,4.451,-51.719,179.783,6.503,149.251
C06125=1113.735,4.202,-51.705,179.783,6.499,149.250
C06126=1113.740,3.952,-51.691,179.782,6.494,149.249
C06127=1113.745,3.702,-51.676,179.781,6.490,149.248
C06128=1113.749,3.453,-51.662,179.781,6.485,149.247
C06129=1113.755,3.204,-51.648,179.780,6.480,149.247
C06130=1113.760,2.954,-51.634,179.780,6.476,149.246
C06131=1113.765,2.704,-51.620,179.779,6.471,149.245
C06132=1113.770,2.455,-51.605,179.778,6.466,149.244
C06133=1113.775,2.205,-51.591,179.778,6.463,149.243
C06134=1113.780,1.956,-51.577,179.778,6.458,149.242
C06135=1113.785,1.706,-51.563,179.777,6.454,149.242
C06136=1113.790,1.457,-51.549,179.776,6.449,149.241
C06137=1113.795,1.207,-51.535,179.776,6.444,149.240
C06138=1113.800,0.958,-51.521,179.775,6.439,149.239
C06139=1113.805,0.708,-51.507,179.774,6.435,149.238
C06140=1113.810,0.459,-51.492,179.774,6.430,149.237
C06141=1113.816,0.209,-51.479,179.773,6.426,149.237
C06142=1113.821,-0.041,-51.465,179.773,6.422,149.236
C06143=1113.826,-0.290,-51.451,179.772,6.417,149.235
C06144=1113.831,-0.540,-51.436,179.772,6.413,149.234
C06145=1113.836,-0.789,-51.423,179.771,6.408,149.233
C06146=1113.840,-1.039,-51.409,179.770,6.404,149.233
C06147=1113.845,-1.288,-51.395,179.770,6.399,149.232
C06148=1113.851,-1.538,-51.381,179.769,6.394,149.231
C06149=1113.856,-1.788,-51.367,179.768,6.389,149.230
C06150=1113.861,-2.037,-51.353,179.767,6.385,149.229
C06151=1113.867,-2.286,-51.339,179.767,6.380,149.228
C06152=1113.871,-2.536,-51.325,179.767,6.376,149.227
C06153=1113.876,-2.786,-51.312,179.766,6.372,149.227
C06154=1113.882,-3.035,-51.298,179.766,6.367,149.226
C06155=1113.887,-3.285,-51.283,179.765,6.363,149.225
C06156=1113.892,-3.534,-51.269,179.764,6.358,149.224
C06157=1113.896,-3.749,-51.258,179.764,6.354,149.223
C06158=1113.900,-3.964,-51.245,179.763,6.350,149.223
C06159=1113.905,-4.178,-51.234,179.763,6.347,149.222
C06160=1113.909,-4.393,-51.222,179.762,6.343,149.221
C06161=1113.914,-4.607,-51.210,179.761,6.339,149.221
C06162=1113.918,-4.821,-51.198,179.761,6.335,149.220
C06163=1113.922,-5.037,-51.187,179.761,6.331,149.219
C06164=1113.927,-5.250,-51.175,179.760,6.327,149.219
C06165=1113.932,-5.501,-51.161,179.759,6.322,149.218
C06166=1113.936,-5.750,-51.147,179.758,6.318,149.217
C06167=1113.942,-5.999,-51.134,179.759,6.314,149.216
C06168=1113.947,-6.250,-51.120,179.758,6.309,149.215
C06169=1113.952,-6.498,-51.107,179.757,6.305,149.215
C06170=1113.957,-6.748,-51.092,179.757,6.300,149.214
C06171=1113.962,-6.998,-51.079,179.756,6.295,149.213
C06172=1113.968,-7.247,-51.065,179.756,6.291,149.212
C06173=1113.972,-7.497,-51.052,179.755,6.286,149.211
C06174=1113.978,-7.746,-51.038,179.754,6.282,149.210
C06175=1113.983,-7.997,-51.024,179.754,6.277,149.209
C06176=1113.987,-8.246,-51.011,179.753,6.273,149.209
C06177=1113.993,-8.495,-50.997,179.753,6.269,149.208
C06178=1113.998,-8.745,-50.983,179.752,6.264,149.207
C06179=1114.003,-8.994,-50.970,179.752,6.259,149.206
C06180=1114.008,-9.244,-50.956,179.751,6.255,149.205
C06181=1114.014,-9.493,-50.942,179.750,6.250,149.205
C06182=1114.018,-9.743,-50.930,179.750,6.245,149.204
C06183=1114.024,-9.992,-50.916,179.749,6.241,149.203
C06184=1114.028,-10.243,-50.903,179.748,6.236,149.202
C06185=1114.033,-10.492,-50.888,179.748,6.232,149.201
C06186=1114.039,-10.742,-50.875,179.747,6.227,149.200
C06187=1114.043,-10.991,-50.861,179.746,6.223,149.200
C06188=1114.049,-11.241,-50.848,179.746,6.218,149.199
C06189=1114.053,-11.490,-50.835,179.746,6.214,149.198
C06190=1114.059,-11.740,-50.821,179.745,6.209,149.197
C06191=1114.064,-11.990,-50.808,179.744,6.205,149.196
C06192=1114.069,-12.239,-50.795,179.744,6.200,149.195
C06193=1114.075,-12.489,-50.781,179.743,6.195,149.194
C06194=1114.079,-12.738,-50.768,179.743,6.191,149.194
C06195=1114.085,-12.988,-50.754,179.742,6.186,149.193
C06196=1114.090,-13.238,-50.742,179.741,6.182,149.192
C06197=1114.095,-13.487,-50.727,179.741,6.177,149.191
C06198=1114.100,-13.737,-50.715,179.740,6.172,149.190
C06199=1114.105,-13.987,-50.701,179.739,6.168,149.190
C06200=1114.110,-14.236,-50.688,179.739,6.163,149.189
C06201=1114.115,-14.486,-50.674,179.738,6.158,149.188
C06202=1114.120,-14.735,-50.662,179.738,6.154,149.187
C06203=1114.126,-14.984,-50.648,179.737,6.149,149.186
C06204=1114.130,-15.234,-50.635,179.736,6.145,149.185
C06205=1114.136,-15.484,-50.622,179.736,6.141,149.184
C06206=1114.141,-15.733,-50.608,179.736,6.136,149.184
C06207=1114.146,-15.983,-50.595,179.735,6.131,149.183
C06208=1114.151,-16.233,-50.582,179.735,6.126,149.182
C06209=1114.156,-16.482,-50.569,179.734,6.122,149.181
C06210=1114.161,-16.732,-50.555,179.733,6.117,149.180
C06211=1114.166,-16.981,-50.542,179.733,6.113,149.179
C06212=1114.172,-17.231,-50.529,179.732,6.108,149.178
C06213=1114.175,-17.446,-50.518,179.732,6.104,149.178
C06214=1114.180,-17.660,-50.507,179.731,6.100,149.177
C06215=1114.185,-17.875,-50.495,179.731,6.096,149.176
C06216=1114.190,-18.090,-50.484,179.730,6.092,149.175
C06217=1114.193,-18.305,-50.473,179.730,6.088,149.175
C06218=1114.198,-18.519,-50.462,179.729,6.084,149.174
C06219=1114.203,-18.734,-50.450,179.729,6.080,149.173
C06220=1114.207,-18.949,-50.439,179.728,6.076,149.173
C06221=1114.212,-19.198,-50.425,179.728,6.071,149.172
C06222=1114.217,-19.447,-50.413,179.727,6.066,149.171
C06223=1114.222,-19.697,-50.399,179.727,6.061,149.170
C06224=1114.227,-19.947,-50.386,179.726,6.057,149.169
C06225=1114.232,-20.196,-50.374,179.726,6.052,149.168
C06226=1114.238,-20.446,-50.360,179.725,6.047,149.167
C06227=1114.243,-20.696,-50.348,179.725,6.043,149.166
C06228=1114.248,-20.945,-50.335,179.724,6.038,149.165
C06229=1114.253,-21.195,-50.322,179.723,6.033,149.165
C06230=1114.258,-21.444,-50.309,179.723,6.029,149.164
C06231=1114.263,-21.694,-50.296,179.722,6.024,149.163
C06232=1114.268,-21.944,-50.282,179.722,6.019,149.162
C06233=1114.273,-22.193,-50.269,179.721,6.015,149.161
C06234=1114.279,-22.442,-50.257,179.721,6.010,149.160
C06235=1114.284,-22.692,-50.243,179.720,6.005,149.159
C06236=1114.289,-22.942,-50.231,179.720,6.000,149.158
C06237=1114.294,-23.191,-50.218,179.719,5.996,149.158
C06238=1114.299,-23.441,-50.205,179.719,5.991,149.157
C06239=1114.304,-23.691,-50.192,179.718,5.986,149.156
C06240=1114.310,-23.940,-50.179,179.718,5.981,149.155
C06241=1114.315,-24.190,-50.167,179.718,5.977,149.154
C06242=1114.320,-24.440,-50.154,179.717,5.972,149.153
C06243=1114.325,-24.690,-50.141,179.717,5.967,149.152
C06244=1114.331,-24.939,-50.129,179.716,5.962,149.151
C06245=1114.336,-25.188,-50.116,179.716,5.958,149.150
C06246=1114.340,-25.438,-50.103,179.715,5.953,149.149
C06247=1114.346,-25.688,-50.090,179.715,5.948,149.149
C06248=1114.351,-25.937,-50.077,179.715,5.943,149.147
C06249=1114.356,-26.187,-50.064,179.715,5.939,149.146
C06250=1114.361,-26.437,-50.052,179.715,5.935,149.145
C06251=1114.366,-26.686,-50.039,179.716,5.931,149.144
C06252=1114.371,-26.936,-50.027,179.716,5.926,149.143
C06253=1114.377,-27.186,-50.014,179.716,5.921,149.142
C06254=1114.382,-27.436,-50.001,179.716,5.918,149.141
C06255=1114.387,-27.685,-49.989,179.717,5.913,149.140
C06256=1114.392,-27.934,-49.976,179.716,5.908,149.139
C06257=1114.397,-28.183,-49.963,179.717,5.904,149.138
C06258=1114.402,-28.434,-49.951,179.717,5.900,149.137
C06259=1114.407,-28.683,-49.938,179.717,5.896,149.136
C06260=1114.413,-28.933,-49.925,179.717,5.891,149.135
C06261=1114.417,-29.149,-49.914,179.717,5.888,149.134
C06262=1114.422,-29.365,-49.903,179.718,5.884,149.134
C06263=1114.426,-29.581,-49.892,179.718,5.881,149.133
C06264=1114.431,-29.797,-49.881,179.718,5.877,149.132
C06265=1114.435,-30.013,-49.870,179.718,5.873,149.131
C06266=1114.439,-30.229,-49.860,179.717,5.870,149.130
C06267=1114.443,-30.445,-49.849,179.718,5.866,149.130
C06268=1114.448,-30.661,-49.838,179.718,5.862,149.129
C06269=1114.453,-30.909,-49.826,179.717,5.857,149.128
C06270=1114.459,-31.158,-49.813,179.717,5.853,149.127
C06271=1114.463,-31.406,-49.801,179.717,5.848,149.126
C06272=1114.469,-31.655,-49.788,179.717,5.844,149.125
C06273=1114.473,-31.902,-49.776,179.717,5.840,149.124
C06274=1114.479,-32.151,-49.764,179.717,5.836,149.123
C06275=1114.484,-32.400,-49.750,179.716,5.831,149.122
C06276=1114.489,-32.648,-49.739,179.716,5.827,149.122
C06277=1114.494,-32.897,-49.726,179.715,5.823,149.121
C06278=1114.499,-33.147,-49.714,179.715,5.818,149.120
C06279=1114.505,-33.397,-49.702,179.715,5.814,149.119
C06280=1114.510,-33.646,-49.689,179.715,5.809,149.118
C06281=1114.514,-33.897,-49.677,179.714,5.804,149.117
C06282=1114.520,-34.146,-49.664,179.714,5.800,149.116
C06283=1114.525,-34.395,-49.652,179.713,5.795,149.115
C06284=1114.531,-34.645,-49.639,179.713,5.791,149.115
C06285=1114.536,-34.895,-49.627,179.713,5.787,149.114
C06286=1114.540,-35.144,-49.615,179.712,5.782,149.113
C06287=1114.546,-35.394,-49.603,179.712,5.777,149.112
C06288=1114.551,-35.643,-49.590,179.711,5.773,149.111
C06289=1114.556,-35.894,-49.578,179.710,5.768,149.110
C06290=1114.561,-36.143,-49.565,179.710,5.763,149.109
C06291=1114.566,-36.392,-49.553,179.709,5.759,149.108
C06292=1114.571,-36.642,-49.541,179.708,5.754,149.108
C06293=1114.577,-36.892,-49.528,179.708,5.750,149.107
C06294=1114.582,-37.141,-49.516,179.707,5.745,149.106
C06295=1114.587,-37.391,-49.504,179.707,5.740,149.105
C06296=1114.593,-37.641,-49.492,179.706,5.736,149.104
C06297=1114.598,-37.890,-49.479,179.705,5.730,149.103
C06298=1114.603,-38.140,-49.467,179.705,5.725,149.103
C06299=1114.608,-38.389,-49.455,179.704,5.721,149.102
C06300=1114.614,-38.639,-49.443,179.703,5.716,149.101
C06301=1114.619,-38.889,-49.430,179.702,5.711,149.100
C06302=1114.624,-39.138,-49.418,179.702,5.706,149.099
C06303=1114.629,-39.388,-49.407,179.701,5.702,149.099
C06304=1114.633,-39.638,-49.394,179.700,5.696,149.098
C06305=1114.639,-39.888,-49.382,179.699,5.691,149.097
C06306=1114.644,-40.137,-49.370,179.698,5.686,149.096
C06307=1114.649,-40.387,-49.358,179.697,5.681,149.095
C06308=1114.655,-40.637,-49.345,179.696,5.676,149.094
C06309=1114.660,-40.887,-49.333,179.696,5.671,149.093
C06310=1114.665,-41.136,-49.322,179.695,5.666,149.092
C06311=1114.670,-41.385,-49.309,179.694,5.661,149.092
C06312=1114.675,-41.635,-49.297,179.693,5.656,149.091
C06313=1114.681,-41.885,-49.286,179.692,5.650,149.090
C06314=1114.686,-42.134,-49.273,179.691,5.645,149.089
C06315=1114.691,-42.384,-49.262,179.690,5.640,149.088
C06316=1114.696,-42.634,-49.250,179.689,5.634,149.087
C06317=1114.702,-42.883,-49.238,179.688,5.629,149.087
C06318=1114.707,-43.133,-49.226,179.688,5.624,149.085
C06319=1114.712,-43.382,-49.214,179.689,5.620,149.084
C06320=1114.717,-43.632,-49.202,179.688,5.615,149.083
C06321=1114.722,-43.882,-49.190,179.688,5.610,149.082
C06322=1114.728,-44.132,-49.178,179.689,5.606,149.081
C06323=1114.732,-44.381,-49.167,179.689,5.600,149.080
C06324=1114.738,-44.631,-49.155,179.689,5.596,149.079
C06325=1114.742,-44.846,-49.145,179.689,5.591,149.078
C06326=1114.747,-45.061,-49.135,179.689,5.587,149.077
C06327=1114.751,-45.275,-49.123,179.689,5.583,149.076
C06328=1114.756,-45.490,-49.113,179.690,5.580,149.075
C06329=1114.760,-45.705,-49.103,179.690,5.576,149.074
C06330=1114.764,-45.920,-49.093,179.690,5.572,149.073
C06331=1114.769,-46.135,-49.083,179.690,5.568,149.072
C06332=1114.773,-46.350,-49.073,179.690,5.564,149.071
C06333=1114.778,-46.600,-49.062,179.690,5.559,149.070
C06334=1114.784,-46.849,-49.050,179.690,5.554,149.069
C06335=1114.790,-47.098,-49.037,179.691,5.550,149.068
C06336=1114.794,-47.348,-49.026,179.691,5.544,149.067
C06337=1114.800,-47.598,-49.014,179.691,5.540,149.066
C06338=1114.804,-47.847,-49.003,179.691,5.535,149.065
C06339=1114.810,-48.097,-48.991,179.691,5.530,149.064
C06340=1114.815,-48.347,-48.979,179.692,5.526,149.063
C06341=1114.820,-48.597,-48.968,179.691,5.521,149.062
C06342=1114.825,-48.847,-48.956,179.692,5.517,149.061
C06343=1114.831,-49.096,-48.945,179.692,5.512,149.060
C06344=1114.836,-49.345,-48.933,179.692,5.507,149.058
C06345=1114.841,-49.595,-48.921,179.692,5.503,149.057
C06346=1114.847,-49.845,-48.909,179.692,5.497,149.056
C06347=1114.851,-50.095,-48.897,179.693,5.493,149.055
C06348=1114.857,-50.345,-48.886,179.693,5.488,149.054
C06349=1114.861,-50.594,-48.874,179.693,5.483,149.053
C06350=1114.867,-50.843,-48.863,179.693,5.479,149.052
C06351=1114.873,-51.093,-48.851,179.693,5.474,149.051
C06352=1114.878,-51.343,-48.840,179.693,5.469,149.050
C06353=1114.883,-51.593,-48.828,179.694,5.465,149.049
C06354=1114.888,-51.843,-48.816,179.693,5.460,149.048
C06355=1114.893,-52.093,-48.805,179.694,5.456,149.047
C06356=1114.898,-52.341,-48.794,179.694,5.450,149.045
C06357=1114.904,-52.591,-48.782,179.694,5.446,149.045
C06358=1114.909,-52.841,-48.770,179.694,5.441,149.043
C06359=1114.914,-53.091,-48.759,179.694,5.436,149.042
C06360=1114.919,-53.341,-48.747,179.695,5.432,149.041
C06361=1114.925,-53.590,-48.736,179.695,5.427,149.040
C06362=1114.930,-53.840,-48.724,179.695,5.422,149.039
C06363=1114.935,-54.089,-48.713,179.695,5.418,149.038
C06364=1114.940,-54.339,-48.701,179.695,5.413,149.037
C06365=1114.945,-54.589,-48.689,179.696,5.409,149.036
C06366=1114.951,-54.839,-48.679,179.695,5.404,149.035
C06367=1114.956,-55.088,-48.667,179.695,5.399,149.034
C06368=1114.961,-55.338,-48.655,179.696,5.394,149.033
C06369=1114.966,-55.588,-48.644,179.696,5.390,149.032
C06370=1114.972,-55.838,-48.632,179.696,5.384,149.031
C06371=1114.977,-56.087,-48.621,179.696,5.380,149.029
C06372=1114.982,-56.336,-48.610,179.696,5.375,149.028
C06373=1114.987,-56.586,-48.598,179.697,5.371,149.027
C06374=1114.992,-56.836,-48.587,179.697,5.366,149.026
C06375=1114.998,-57.086,-48.576,179.696,5.361,149.025
C06376=1115.003,-57.335,-48.565,179.697,5.357,149.024
C06377=1115.008,-57.585,-48.553,179.697,5.352,149.023
C06378=1115.013,-57.835,-48.542,179.697,5.348,149.022
C06379=1115.018,-58.084,-48.531,179.698,5.343,149.021
C06380=1115.024,-58.334,-48.519,179.697,5.338,149.020
C06381=1115.028,-58.549,-48.509,179.697,5.334,149.019
C06382=1115.033,-58.764,-48.499,179.698,5.330,149.018
C06383=1115.037,-58.979,-48.489,179.698,5.326,149.017
C06384=1115.042,-59.194,-48.481,179.698,5.322,149.016
C06385=1115.046,-59.409,-48.471,179.698,5.318,149.015
C06386=1115.051,-59.624,-48.461,179.698,5.314,149.014
C06387=1115.054,-59.838,-48.451,179.699,5.310,149.013
C06388=1115.059,-60.054,-48.442,179.699,5.306,149.013
C06389=1115.065,-60.303,-48.430,179.698,5.301,149.012
C06390=1115.070,-60.553,-48.419,179.697,5.296,149.011
C06391=1115.074,-60.802,-48.408,179.696,5.290,149.010
C06392=1115.080,-61.053,-48.397,179.696,5.286,149.009
C06393=1115.085,-61.302,-48.386,179.696,5.280,149.008
C06394=1115.091,-61.552,-48.374,179.695,5.275,149.007
C06395=1115.096,-61.802,-48.363,179.695,5.270,149.006
C06396=1115.101,-62.051,-48.352,179.694,5.265,149.005
C06397=1115.106,-62.300,-48.341,179.693,5.260,149.004
C06398=1115.112,-62.551,-48.330,179.693,5.255,149.003
C06399=1115.117,-62.800,-48.319,179.693,5.250,149.002
C06400=1115.122,-63.049,-48.308,179.692,5.244,149.001
C06401=1115.127,-63.300,-48.296,179.692,5.240,149.000
C06402=1115.133,-63.549,-48.285,179.692,5.235,148.999
C06403=1115.137,-63.799,-48.274,179.691,5.229,148.998
C06404=1115.143,-64.049,-48.263,179.690,5.224,148.997
C06405=1115.148,-64.298,-48.252,179.691,5.219,148.996
C06406=1115.153,-64.548,-48.242,179.690,5.213,148.995
C06407=1115.159,-64.797,-48.231,179.689,5.209,148.994
C06408=1115.164,-65.048,-48.219,179.689,5.204,148.993
C06409=1115.169,-65.297,-48.208,179.688,5.198,148.992
C06410=1115.175,-65.547,-48.198,179.688,5.193,148.991
C06411=1115.179,-65.797,-48.187,179.688,5.188,148.990
C06412=1115.185,-66.045,-48.176,179.687,5.183,148.989
C06413=1115.190,-66.296,-48.165,179.687,5.177,148.988
C06414=1115.195,-66.546,-48.153,179.687,5.173,148.987
C06415=1115.201,-66.795,-48.143,179.686,5.167,148.986
C06416=1115.205,-67.045,-48.132,179.686,5.162,148.985
C06417=1115.211,-67.294,-48.122,179.686,5.157,148.984
C06418=1115.217,-67.545,-48.110,179.686,5.152,148.983
C06419=1115.222,-67.794,-48.099,179.685,5.146,148.982
C06420=1115.227,-68.044,-48.089,179.685,5.141,148.980
C06421=1115.232,-68.294,-48.078,179.685,5.136,148.980
C06422=1115.237,-68.543,-48.067,179.685,5.131,148.978
C06423=1115.242,-68.793,-48.056,179.684,5.125,148.977
C06424=1115.248,-69.043,-48.045,179.684,5.120,148.976
C06425=1115.253,-69.293,-48.035,179.684,5.115,148.975
C06426=1115.259,-69.542,-48.024,179.684,5.110,148.974
C06427=1115.264,-69.792,-48.013,179.684,5.104,148.973
C06428=1115.269,-70.041,-48.002,179.684,5.099,148.972
C06429=1115.274,-70.291,-47.992,179.683,5.095,148.971
C06430=1115.279,-70.541,-47.982,179.684,5.089,148.970
C06431=1115.284,-70.791,-47.970,179.683,5.083,148.969
C06432=1115.290,-71.040,-47.960,179.683,5.079,148.968
C06433=1115.295,-71.290,-47.949,179.683,5.074,148.967
C06434=1115.301,-71.540,-47.939,179.683,5.068,148.965
C06435=1115.306,-71.790,-47.927,179.683,5.063,148.964
C06436=1115.311,-72.039,-47.917,179.683,5.059,148.963
C06437=1115.315,-72.255,-47.908,179.682,5.054,148.962
C06438=1115.320,-72.469,-47.898,179.683,5.049,148.961
C06439=1115.325,-72.684,-47.890,179.683,5.045,148.960
C06440=1115.329,-72.899,-47.881,179.682,5.040,148.959
C06441=1115.334,-73.114,-47.872,179.683,5.036,148.958
C06442=1115.339,-73.330,-47.863,179.682,5.031,148.957
C06443=1115.342,-73.544,-47.853,179.682,5.026,148.956
C06444=1115.348,-73.759,-47.844,179.682,5.022,148.956
C06445=1115.353,-74.009,-47.834,179.682,5.017,148.954
C06446=1115.358,-74.259,-47.823,179.682,5.012,148.953
C06447=1115.363,-74.509,-47.813,179.682,5.006,148.952
C06448=1115.368,-74.758,-47.802,179.682,5.001,148.951
C06449=1115.374,-75.007,-47.792,179.682,4.996,148.950
C06450=1115.379,-75.258,-47.781,179.682,4.991,148.949
C06451=1115.385,-75.507,-47.771,179.682,4.986,148.948
C06452=1115.390,-75.757,-47.760,179.682,4.981,148.946
C06453=1115.395,-76.007,-47.750,179.682,4.976,148.945
C06454=1115.400,-76.256,-47.739,179.683,4.971,148.944
C06455=1115.405,-76.506,-47.729,179.683,4.965,148.943
C06456=1115.411,-76.756,-47.719,179.683,4.960,148.942
C06457=1115.416,-77.006,-47.708,179.683,4.955,148.941
C06458=1115.422,-77.256,-47.698,179.683,4.950,148.939
C06459=1115.427,-77.505,-47.688,179.683,4.944,148.938
C06460=1115.432,-77.755,-47.678,179.683,4.939,148.937
C06461=1115.437,-78.005,-47.667,179.683,4.934,148.936
C06462=1115.442,-78.255,-47.657,179.683,4.929,148.935
C06463=1115.448,-78.504,-47.647,179.683,4.923,148.934
C06464=1115.453,-78.753,-47.636,179.683,4.918,148.932
C06465=1115.458,-79.003,-47.625,179.684,4.913,148.931
C06466=1115.464,-79.253,-47.615,179.684,4.908,148.930
C06467=1115.469,-79.503,-47.605,179.684,4.903,148.929
C06468=1115.474,-79.753,-47.594,179.684,4.898,148.928
C06469=1115.479,-80.002,-47.584,179.684,4.892,148.927
C06470=1115.485,-80.252,-47.574,179.684,4.887,148.925
C06471=1115.490,-80.502,-47.564,179.685,4.882,148.924
C06472=1115.495,-80.751,-47.553,179.685,4.878,148.923
C06473=1115.501,-81.001,-47.543,179.686,4.873,148.922
C06474=1115.506,-81.251,-47.533,179.686,4.868,148.921
C06475=1115.511,-81.500,-47.523,179.686,4.862,148.920
C06476=1115.517,-81.751,-47.514,179.686,4.857,148.918
C06477=1115.522,-82.001,-47.503,179.686,4.852,148.917
C06478=1115.527,-82.250,-47.493,179.687,4.847,148.916
C06479=1115.533,-82.500,-47.483,179.687,4.841,148.915
C06480=1115.538,-82.749,-47.472,179.687,4.836,148.913
C06481=1115.543,-82.999,-47.462,179.687,4.831,148.912
C06482=1115.548,-83.249,-47.452,179.688,4.826,148.911
C06483=1115.554,-83.498,-47.442,179.688,4.822,148.910
C06484=1115.559,-83.749,-47.431,179.688,4.816,148.909
C06485=1115.564,-83.998,-47.422,179.689,4.811,148.908
C06486=1115.569,-84.247,-47.412,179.689,4.806,148.906
C06487=1115.575,-84.498,-47.402,179.690,4.801,148.905
C06488=1115.580,-84.748,-47.391,179.690,4.795,148.904
C06489=1115.585,-84.997,-47.382,179.690,4.791,148.903
C06490=1115.591,-85.247,-47.372,179.691,4.786,148.901
C06491=1115.596,-85.497,-47.361,179.691,4.781,148.900
C06492=1115.601,-85.746,-47.351,179.691,4.776,148.899
C06493=1115.606,-85.961,-47.343,179.692,4.771,148.898
C06494=1115.610,-86.177,-47.335,179.692,4.767,148.897
C06495=1115.615,-86.392,-47.326,179.692,4.763,148.896
C06496=1115.619,-86.607,-47.317,179.692,4.758,148.895
C06497=1115.624,-86.821,-47.308,179.693,4.754,148.894
C06498=1115.628,-87.037,-47.299,179.693,4.750,148.893
C06499=1115.633,-87.252,-47.292,179.693,4.745,148.892
C06500=1115.638,-87.467,-47.282,179.694,4.741,148.891
C06501=1115.643,-87.716,-47.273,179.695,4.736,148.889
C06502=1115.648,-87.966,-47.263,179.695,4.731,148.888
C06503=1115.654,-88.217,-47.253,179.695,4.726,148.887
C06504=1115.658,-88.466,-47.243,179.695,4.721,148.886
C06505=1115.664,-88.716,-47.233,179.696,4.717,148.885
C06506=1115.670,-88.965,-47.223,179.697,4.711,148.883
C06507=1115.675,-89.215,-47.214,179.697,4.706,148.882
C06508=1115.680,-89.465,-47.203,179.698,4.702,148.881
C06509=1115.685,-89.715,-47.193,179.698,4.696,148.880
C06510=1115.690,-89.964,-47.183,179.699,4.692,148.878
C06511=1115.696,-90.214,-47.174,179.699,4.687,148.877
C06512=1115.701,-90.463,-47.164,179.700,4.681,148.876
C06513=1115.706,-90.714,-47.154,179.700,4.677,148.875
C06514=1115.712,-90.964,-47.144,179.701,4.672,148.874
C06515=1115.717,-91.213,-47.135,179.701,4.668,148.872
C06516=1115.722,-91.463,-47.124,179.702,4.662,148.871
C06517=1115.728,-91.713,-47.115,179.702,4.657,148.870
C06518=1115.733,-91.962,-47.105,179.703,4.653,148.869
C06519=1115.738,-92.212,-47.095,179.703,4.647,148.867
C06520=1115.743,-92.462,-47.086,179.704,4.643,148.866
C06521=1115.749,-92.712,-47.076,179.704,4.638,148.865
C06522=1115.754,-92.962,-47.067,179.705,4.634,148.864
C06523=1115.760,-93.211,-47.057,179.705,4.628,148.863
C06524=1115.765,-93.461,-47.046,179.706,4.624,148.861
C06525=1115.770,-93.711,-47.037,179.707,4.618,148.860
C06526=1115.775,-93.961,-47.027,179.707,4.614,148.859
C06527=1115.780,-94.210,-47.017,179.708,4.609,148.858
C06528=1115.786,-94.460,-47.008,179.708,4.605,148.856
C06529=1115.791,-94.709,-46.998,179.709,4.599,148.855
C06530=1115.797,-94.959,-46.989,179.709,4.594,148.854
C06531=1115.803,-95.209,-46.978,179.710,4.590,148.853
C06532=1115.808,-95.459,-46.970,179.710,4.585,148.852
C06533=1115.813,-95.709,-46.959,179.710,4.580,148.850
C06534=1115.818,-95.959,-46.950,179.710,4.574,148.849
C06535=1115.823,-96.209,-46.940,179.711,4.570,148.848
C06536=1115.828,-96.458,-46.930,179.711,4.565,148.847
C06537=1115.834,-96.708,-46.921,179.711,4.560,148.846
C06538=1115.839,-96.957,-46.911,179.712,4.555,148.845
C06539=1115.845,-97.207,-46.902,179.712,4.551,148.844
C06540=1115.850,-97.457,-46.892,179.712,4.546,148.842
C06541=1115.856,-97.707,-46.883,179.712,4.540,148.841
C06542=1115.861,-97.956,-46.873,179.713,4.535,148.840
C06543=1115.866,-98.207,-46.863,179.713,4.531,148.839
C06544=1115.871,-98.457,-46.854,179.714,4.526,148.838
C06545=1115.877,-98.706,-46.844,179.714,4.521,148.836
C06546=1115.882,-98.956,-46.835,179.714,4.515,148.835
C06547=1115.887,-99.205,-46.825,179.715,4.511,148.834
C06548=1115.893,-99.455,-46.816,179.715,4.506,148.833
C06549=1115.897,-99.670,-46.808,179.715,4.502,148.832
C06550=1115.901,-99.886,-46.800,179.716,4.497,148.831
C06551=1115.906,-100.100,-46.791,179.716,4.493,148.830
C06552=1115.911,-100.316,-46.783,179.716,4.489,148.829
C06553=1115.916,-100.531,-46.775,179.716,4.485,148.828
C06554=1115.920,-100.746,-46.767,179.717,4.480,148.827
C06555=1115.925,-100.961,-46.759,179.717,4.476,148.826
C06556=1115.929,-101.176,-46.750,179.717,4.472,148.825
C06557=1115.935,-101.426,-46.741,179.718,4.467,148.824
C06558=1115.940,-101.676,-46.732,179.718,4.461,148.822
C06559=1115.945,-101.925,-46.722,179.718,4.456,148.821
C06560=1115.951,-102.176,-46.713,179.719,4.452,148.820
C06561=1115.956,-102.425,-46.704,179.719,4.447,148.819
C06562=1115.961,-102.675,-46.694,179.719,4.442,148.818
C06563=1115.967,-102.925,-46.685,179.719,4.436,148.816
C06564=1115.972,-103.175,-46.676,179.720,4.431,148.815
C06565=1115.977,-103.424,-46.666,179.720,4.426,148.814
C06566=1115.983,-103.674,-46.657,179.721,4.422,148.813
C06567=1115.988,-103.924,-46.648,179.721,4.417,148.812
C06568=1115.993,-104.173,-46.638,179.721,4.411,148.810
C06569=1115.998,-104.423,-46.629,179.721,4.406,148.809
C06570=1116.004,-104.673,-46.620,179.722,4.401,148.808
C06571=1116.010,-104.923,-46.611,179.722,4.396,148.807
C06572=1116.014,-105.173,-46.601,179.723,4.392,148.806
C06573=1116.020,-105.422,-46.592,179.723,4.386,148.804
C06574=1116.025,-105.673,-46.583,179.723,4.381,148.803
C06575=1116.031,-105.922,-46.574,179.723,4.376,148.802
C06576=1116.035,-106.172,-46.564,179.724,4.371,148.801
C06577=1116.041,-106.421,-46.555,179.724,4.366,148.800
C06578=1116.047,-106.672,-46.546,179.724,4.361,148.798
C06579=1116.052,-106.921,-46.537,179.725,4.356,148.797
C06580=1116.057,-107.171,-46.527,179.725,4.351,148.796
C06581=1116.062,-107.421,-46.518,179.725,4.346,148.795
C06582=1116.068,-107.671,-46.509,179.726,4.341,148.794
C06583=1116.073,-107.920,-46.500,179.726,4.336,148.792
C06584=1116.079,-108.170,-46.491,179.726,4.330,148.791
C06585=1116.084,-108.420,-46.482,179.726,4.325,148.790
C06586=1116.089,-108.669,-46.472,179.727,4.320,148.789
C06587=1116.095,-108.919,-46.463,179.727,4.315,148.788
C06588=1116.100,-109.169,-46.454,179.727,4.310,148.786
C06589=1116.105,-109.419,-46.446,179.728,4.305,148.785
C06590=1116.111,-109.669,-46.436,179.728,4.300,148.784
C06591=1116.116,-109.919,-46.427,179.729,4.295,148.783
C06592=1116.121,-110.169,-46.418,179.729,4.290,148.782
C06593=1116.126,-110.418,-46.409,179.729,4.285,148.780
C06594=1116.132,-110.668,-46.401,179.729,4.280,148.779
C06595=1116.138,-110.917,-46.391,179.730,4.274,148.778
C06596=1116.143,-111.167,-46.382,179.730,4.269,148.777
C06597=1116.148,-111.417,-46.373,179.730,4.264,148.776
C06598=1116.153,-111.667,-46.364,179.730,4.259,148.774
C06599=1116.158,-111.916,-46.355,179.731,4.254,148.773
C06600=1116.163,-112.166,-46.346,179.731,4.249,148.772
C06601=1116.169,-112.417,-46.337,179.731,4.243,148.771
C06602=1116.175,-112.666,-46.328,179.731,4.238,148.770
C06603=1116.180,-112.916,-46.319,179.732,4.233,148.768
C06604=1116.185,-113.165,-46.310,179.732,4.228,148.767
C06605=1116.190,-113.380,-46.303,179.733,4.224,148.766
C06606=1116.194,-113.596,-46.295,179.733,4.220,148.765
C06607=1116.199,-113.811,-46.287,179.733,4.215,148.764
C06608=1116.204,-114.026,-46.279,179.734,4.211,148.763
C06609=1116.209,-114.242,-46.272,179.733,4.206,148.762
C06610=1116.213,-114.457,-46.264,179.734,4.201,148.761
C06611=1116.218,-114.672,-46.256,179.734,4.197,148.760
C06612=1116.222,-114.887,-46.249,179.734,4.193,148.759
C06613=1116.228,-115.137,-46.240,179.735,4.187,148.757
C06614=1116.233,-115.387,-46.231,179.735,4.182,148.756
C06615=1116.239,-115.636,-46.222,179.736,4.177,148.755
C06616=1116.244,-115.886,-46.213,179.736,4.172,148.754
C06617=1116.249,-116.136,-46.205,179.736,4.166,148.752
C06618=1116.254,-116.386,-46.196,179.736,4.161,148.751
C06619=1116.260,-116.636,-46.187,179.737,4.156,148.750
C06620=1116.266,-116.886,-46.179,179.737,4.151,148.749
C06621=1116.271,-117.135,-46.170,179.737,4.146,148.748
C06622=1116.276,-117.385,-46.161,179.738,4.140,148.746
C06623=1116.281,-117.635,-46.152,179.738,4.135,148.745
C06624=1116.286,-117.885,-46.143,179.738,4.129,148.744
C06625=1116.292,-118.134,-46.135,179.738,4.124,148.743
C06626=1116.298,-118.385,-46.127,179.739,4.119,148.741
C06627=1116.303,-118.634,-46.118,179.739,4.114,148.740
C06628=1116.308,-118.884,-46.109,179.739,4.108,148.739
C06629=1116.314,-119.133,-46.100,179.740,4.103,148.737
C06630=1116.319,-119.383,-46.091,179.740,4.098,148.736
C06631=1116.324,-119.633,-46.083,179.740,4.092,148.735
C06632=1116.329,-119.884,-46.074,179.741,4.087,148.734
C06633=1116.335,-120.133,-46.066,179.741,4.082,148.733
C06634=1116.340,-120.383,-46.057,179.741,4.077,148.731
C06635=1116.346,-120.632,-46.048,179.742,4.071,148.730
C06636=1116.352,-120.882,-46.040,179.742,4.065,148.729
C06637=1116.357,-121.132,-46.031,179.742,4.060,148.728
C06638=1116.362,-121.382,-46.022,179.742,4.055,148.726
C06639=1116.367,-121.632,-46.013,179.743,4.050,148.725
C06640=1116.373,-121.882,-46.006,179.743,4.044,148.724
C06641=1116.378,-122.131,-45.997,179.744,4.039,148.722
C06642=1116.384,-122.381,-45.988,179.744,4.034,148.721
C06643=1116.390,-122.631,-45.980,179.744,4.028,148.720
C06644=1116.395,-122.881,-45.971,179.744,4.023,148.719
C06645=1116.399,-123.130,-45.963,179.745,4.017,148.717
C06646=1116.404,-123.380,-45.954,179.745,4.012,148.716
C06647=1116.410,-123.630,-45.946,179.745,4.007,148.715
C06648=1116.416,-123.880,-45.937,179.746,4.002,148.714
C06649=1116.421,-124.130,-45.928,179.746,3.995,148.712
C06650=1116.427,-124.379,-45.921,179.746,3.990,148.711
C06651=1116.432,-124.629,-45.912,179.747,3.985,148.710
C06652=1116.437,-124.880,-45.903,179.747,3.980,148.708
C06653=1116.442,-125.129,-45.896,179.748,3.974,148.707
C06654=1116.448,-125.378,-45.887,179.747,3.968,148.706
C06655=1116.454,-125.628,-45.879,179.748,3.963,148.705
C06656=1116.459,-125.878,-45.870,179.748,3.958,148.703
C06657=1116.464,-126.129,-45.862,179.749,3.953,148.702
C06658=1116.470,-126.378,-45.853,179.749,3.947,148.701
C06659=1116.475,-126.627,-45.845,179.749,3.941,148.699
C06660=1116.480,-126.878,-45.837,179.750,3.936,148.698
C06661=1116.485,-127.093,-45.829,179.750,3.931,148.697
C06662=1116.490,-127.309,-45.822,179.750,3.927,148.696
C06663=1116.494,-127.523,-45.815,179.751,3.921,148.695
C06664=1116.499,-127.739,-45.808,179.750,3.917,148.694
C06665=1116.504,-127.954,-45.801,179.751,3.912,148.693
C06666=1116.508,-128.169,-45.794,179.752,3.907,148.691
C06667=1116.513,-128.385,-45.787,179.751,3.902,148.690
C06668=1116.518,-128.600,-45.779,179.752,3.898,148.689
C06669=1116.095,-128.590,-45.806,179.759,3.902,148.688
C06670=1116.090,-128.375,-45.812,179.759,3.907,148.689
C06671=1116.085,-128.160,-45.820,179.759,3.912,148.690
C06672=1116.080,-127.944,-45.827,179.758,3.916,148.691
C06673=1116.076,-127.729,-45.834,179.758,3.921,148.692
C06674=1116.071,-127.514,-45.841,179.758,3.926,148.693
C06675=1116.066,-127.298,-45.848,179.757,3.930,148.695
C06676=1116.062,-127.084,-45.855,179.757,3.935,148.696
C06677=1116.057,-126.869,-45.863,179.757,3.940,148.697
C06678=1116.052,-126.618,-45.871,179.757,3.946,148.698
C06679=1116.046,-126.369,-45.880,179.756,3.951,148.699
C06680=1116.041,-126.118,-45.888,179.755,3.956,148.701
C06681=1116.036,-125.869,-45.896,179.756,3.962,148.702
C06682=1116.030,-125.620,-45.905,179.755,3.967,148.703
C06683=1116.025,-125.369,-45.913,179.755,3.973,148.705
C06684=1116.020,-125.119,-45.922,179.754,3.978,148.706
C06685=1116.014,-124.870,-45.930,179.754,3.983,148.707
C06686=1116.009,-124.620,-45.939,179.754,3.989,148.708
C06687=1116.003,-124.370,-45.947,179.753,3.995,148.710
C06688=1115.998,-124.120,-45.955,179.753,4.000,148.711
C06689=1115.993,-123.871,-45.964,179.753,4.005,148.712
C06690=1115.988,-123.621,-45.972,179.752,4.011,148.714
C06691=1115.982,-123.372,-45.981,179.752,4.016,148.715
C06692=1115.977,-123.121,-45.989,179.752,4.022,148.716
C06693=1115.971,-122.871,-45.998,179.752,4.027,148.717
C06694=1115.966,-122.621,-46.007,179.751,4.033,148.719
C06695=1115.960,-122.372,-46.015,179.751,4.038,148.720
C06696=1115.955,-122.122,-46.024,179.750,4.043,148.721
C06697=1115.950,-121.872,-46.033,179.750,4.048,148.722
C06698=1115.944,-121.623,-46.041,179.750,4.053,148.724
C06699=1115.939,-121.372,-46.049,179.750,4.060,148.725
C06700=1115.933,-121.123,-46.058,179.749,4.065,148.726
C06701=1115.928,-120.873,-46.067,179.749,4.070,148.728
C06702=1115.922,-120.624,-46.076,179.749,4.075,148.729
C06703=1115.918,-120.374,-46.084,179.748,4.080,148.730
C06704=1115.913,-120.123,-46.092,179.748,4.086,148.731
C06705=1115.907,-119.874,-46.101,179.747,4.091,148.733
C06706=1115.902,-119.625,-46.110,179.747,4.096,148.734
C06707=1115.896,-119.375,-46.118,179.747,4.101,148.735
C06708=1115.891,-119.125,-46.127,179.747,4.107,148.736
C06709=1115.886,-118.874,-46.136,179.747,4.113,148.737
C06710=1115.880,-118.625,-46.144,179.746,4.118,148.739
C06711=1115.874,-118.375,-46.154,179.746,4.123,148.740
C06712=1115.869,-118.125,-46.162,179.745,4.129,148.741
C06713=1115.864,-117.875,-46.171,179.745,4.134,148.743
C06714=1115.859,-117.625,-46.180,179.745,4.139,148.744
C06715=1115.853,-117.376,-46.189,179.745,4.144,148.745
C06716=1115.848,-117.126,-46.198,179.744,4.149,148.746
C06717=1115.842,-116.876,-46.206,179.744,4.155,148.748
C06718=1115.837,-116.626,-46.215,179.743,4.160,148.749
C06719=1115.832,-116.376,-46.224,179.743,4.165,148.750
C06720=1115.826,-116.127,-46.232,179.743,4.170,148.751
C06721=1115.821,-115.877,-46.241,179.743,4.175,148.752
C06722=1115.816,-115.627,-46.250,179.742,4.181,148.754
C06723=1115.811,-115.378,-46.259,179.742,4.186,148.755
C06724=1115.805,-115.128,-46.268,179.742,4.191,148.756
C06725=1115.799,-114.878,-46.277,179.741,4.196,148.758
C06726=1115.795,-114.662,-46.285,179.741,4.201,148.758
C06727=1115.791,-114.448,-46.292,179.741,4.205,148.759
C06728=1115.786,-114.233,-46.300,179.740,4.210,148.761
C06729=1115.781,-114.018,-46.307,179.740,4.214,148.762
C06730=1115.777,-113.802,-46.315,179.740,4.218,148.763
C06731=1115.772,-113.587,-46.323,179.740,4.223,148.764
C06732=1115.767,-113.372,-46.330,179.739,4.227,148.765
C06733=1115.762,-113.156,-46.338,179.739,4.233,148.766
C06734=1115.757,-112.907,-46.347,179.739,4.238,148.767
C06735=1115.752,-112.657,-46.356,179.739,4.243,148.768
C06736=1115.746,-112.407,-46.365,179.738,4.247,148.770
C06737=1115.741,-112.157,-46.375,179.737,4.252,148.771
C06738=1115.736,-111.907,-46.384,179.737,4.258,148.772
C06739=1115.730,-111.658,-46.392,179.737,4.263,148.773
C06740=1115.725,-111.408,-46.401,179.737,4.268,148.774
C06741=1115.719,-111.158,-46.411,179.736,4.273,148.776
C06742=1115.714,-110.908,-46.420,179.736,4.278,148.777
C06743=1115.709,-110.659,-46.428,179.736,4.283,148.778
C06744=1115.704,-110.409,-46.437,179.736,4.289,148.779
C06745=1115.699,-110.159,-46.446,179.735,4.294,148.780
C06746=1115.693,-109.909,-46.456,179.735,4.299,148.782
C06747=1115.688,-109.660,-46.465,179.735,4.304,148.783
C06748=1115.683,-109.410,-46.474,179.735,4.309,148.784
C06749=1115.678,-109.160,-46.483,179.734,4.314,148.785
C06750=1115.672,-108.911,-46.492,179.734,4.319,148.786
C06751=1115.666,-108.661,-46.501,179.733,4.324,148.788
C06752=1115.661,-108.411,-46.510,179.733,4.329,148.789
C06753=1115.656,-108.161,-46.520,179.733,4.334,148.790
C06754=1115.650,-107.911,-46.529,179.733,4.339,148.791
C06755=1115.645,-107.661,-46.538,179.732,4.345,148.792
C06756=1115.640,-107.412,-46.547,179.732,4.350,148.794
C06757=1115.634,-107.162,-46.556,179.732,4.355,148.795
C06758=1115.629,-106.912,-46.566,179.732,4.360,148.796
C06759=1115.624,-106.662,-46.575,179.731,4.364,148.797
C06760=1115.618,-106.412,-46.584,179.731,4.370,148.798
C06761=1115.613,-106.162,-46.593,179.730,4.375,148.800
C06762=1115.608,-105.913,-46.603,179.730,4.380,148.801
C06763=1115.603,-105.663,-46.612,179.730,4.385,148.802
C06764=1115.597,-105.413,-46.621,179.730,4.390,148.803
C06765=1115.591,-105.163,-46.630,179.729,4.395,148.804
C06766=1115.587,-104.914,-46.640,179.729,4.400,148.806
C06767=1115.581,-104.664,-46.649,179.728,4.405,148.807
C06768=1115.576,-104.414,-46.658,179.728,4.410,148.808
C06769=1115.571,-104.165,-46.668,179.728,4.415,148.809
C06770=1115.566,-103.915,-46.677,179.728,4.420,148.810
C06771=1115.560,-103.665,-46.686,179.727,4.426,148.812
C06772=1115.555,-103.415,-46.696,179.727,4.430,148.813
C06773=1115.549,-103.165,-46.705,179.726,4.435,148.814
C06774=1115.544,-102.915,-46.714,179.726,4.440,148.815
C06775=1115.539,-102.666,-46.724,179.726,4.445,148.816
C06776=1115.533,-102.416,-46.733,179.726,4.451,148.818
C06777=1115.528,-102.166,-46.742,179.725,4.456,148.819
C06778=1115.523,-101.917,-46.752,179.725,4.460,148.820
C06779=1115.517,-101.667,-46.761,179.724,4.465,148.821
C06780=1115.512,-101.418,-46.771,179.724,4.470,148.822
C06781=1115.506,-101.167,-46.781,179.724,4.476,148.824
C06782=1115.502,-100.952,-46.788,179.724,4.480,148.824
C06783=1115.497,-100.737,-46.797,179.723,4.483,148.825
C06784=1115.493,-100.522,-46.804,179.723,4.489,148.827
C06785=1115.489,-100.307,-46.813,179.723,4.493,148.828
C06786=1115.483,-100.091,-46.821,179.723,4.497,148.829
C06787=1115.479,-99.877,-46.830,179.722,4.501,148.830
C06788=1115.475,-99.661,-46.838,179.722,4.506,148.831
C06789=1115.470,-99.447,-46.846,179.722,4.510,148.832
C06790=1115.464,-99.197,-46.855,179.722,4.515,148.833
C06791=1115.459,-98.947,-46.865,179.721,4.519,148.834
C06792=1115.453,-98.697,-46.875,179.721,4.524,148.835
C06793=1115.448,-98.447,-46.883,179.720,4.529,148.836
C06794=1115.443,-98.197,-46.894,179.720,4.535,148.838
C06795=1115.438,-97.947,-46.903,179.719,4.539,148.839
C06796=1115.432,-97.698,-46.913,179.719,4.544,148.840
C06797=1115.427,-97.448,-46.922,179.719,4.549,148.841
C06798=1115.422,-97.198,-46.932,179.719,4.554,148.842
C06799=1115.417,-96.949,-46.942,179.718,4.559,148.844
C06800=1115.411,-96.699,-46.951,179.718,4.564,148.845
C06801=1115.406,-96.450,-46.961,179.717,4.569,148.846
C06802=1115.400,-96.200,-46.970,179.717,4.574,148.847
C06803=1115.396,-95.950,-46.980,179.717,4.578,148.848
C06804=1115.390,-95.699,-46.990,179.717,4.583,148.849
C06805=1115.385,-95.450,-47.000,179.716,4.589,148.850
C06806=1115.379,-95.200,-47.009,179.716,4.594,148.852
C06807=1115.374,-94.951,-47.019,179.715,4.598,148.853
C06808=1115.369,-94.701,-47.029,179.715,4.603,148.854
C06809=1115.364,-94.451,-47.038,179.715,4.608,148.855
C06810=1115.358,-94.202,-47.048,179.714,4.613,148.856
C06811=1115.353,-93.951,-47.058,179.714,4.618,148.858
C06812=1115.348,-93.702,-47.067,179.713,4.623,148.859
C06813=1115.342,-93.452,-47.078,179.713,4.628,148.860
C06814=1115.337,-93.202,-47.087,179.712,4.632,148.861
C06815=1115.331,-92.953,-47.097,179.712,4.637,148.863
C06816=1115.326,-92.703,-47.107,179.711,4.642,148.864
C06817=1115.321,-92.453,-47.116,179.711,4.647,148.865
C06818=1115.316,-92.203,-47.126,179.710,4.651,148.866
C06819=1115.311,-91.954,-47.136,179.709,4.657,148.868
C06820=1115.305,-91.704,-47.146,179.708,4.661,148.869
C06821=1115.299,-91.454,-47.156,179.708,4.666,148.870
C06822=1115.295,-91.204,-47.166,179.708,4.671,148.871
C06823=1115.289,-90.954,-47.175,179.707,4.676,148.872
C06824=1115.284,-90.705,-47.185,179.707,4.681,148.873
C06825=1115.279,-90.455,-47.195,179.706,4.686,148.875
C06826=1115.273,-90.206,-47.205,179.705,4.691,148.876
C06827=1115.269,-89.955,-47.215,179.705,4.696,148.877
C06828=1115.263,-89.706,-47.225,179.705,4.700,148.878
C06829=1115.257,-89.456,-47.235,179.704,4.705,148.880
C06830=1115.252,-89.207,-47.245,179.704,4.711,148.881
C06831=1115.247,-88.957,-47.254,179.703,4.715,148.882
C06832=1115.242,-88.707,-47.265,179.703,4.720,148.883
C06833=1115.237,-88.457,-47.274,179.702,4.726,148.885
C06834=1115.231,-88.208,-47.284,179.702,4.730,148.886
C06835=1115.225,-87.958,-47.294,179.702,4.735,148.887
C06836=1115.221,-87.708,-47.304,179.701,4.740,148.888
C06837=1115.215,-87.458,-47.314,179.701,4.745,148.889
C06838=1115.210,-87.243,-47.323,179.700,4.750,148.891
C06839=1115.206,-87.028,-47.332,179.700,4.754,148.891
C06840=1115.201,-86.813,-47.339,179.699,4.758,148.893
C06841=1115.197,-86.598,-47.349,179.699,4.762,148.894
C06842=1115.192,-86.383,-47.357,179.699,4.767,148.895
C06843=1115.188,-86.168,-47.366,179.699,4.771,148.896
C06844=1115.183,-85.953,-47.375,179.698,4.775,148.897
C06845=1115.179,-85.738,-47.383,179.698,4.779,148.898
C06846=1115.173,-85.488,-47.393,179.697,4.785,148.899
C06847=1115.168,-85.238,-47.403,179.697,4.790,148.900
C06848=1115.163,-84.988,-47.414,179.697,4.795,148.901
C06849=1115.158,-84.739,-47.423,179.696,4.799,148.903
C06850=1115.152,-84.489,-47.433,179.696,4.805,148.904
C06851=1115.147,-84.240,-47.444,179.695,4.810,148.905
C06852=1115.142,-83.989,-47.454,179.695,4.815,148.906
C06853=1115.137,-83.740,-47.464,179.695,4.820,148.907
C06854=1115.131,-83.491,-47.474,179.695,4.825,148.909
C06855=1115.126,-83.240,-47.485,179.695,4.830,148.910
C06856=1115.120,-82.990,-47.494,179.694,4.835,148.911
C06857=1115.115,-82.741,-47.504,179.694,4.840,148.912
C06858=1115.110,-82.491,-47.514,179.694,4.845,148.913
C06859=1115.105,-82.241,-47.524,179.693,4.851,148.915
C06860=1115.099,-81.992,-47.535,179.693,4.856,148.916
C06861=1115.094,-81.741,-47.545,179.693,4.861,148.917
C06862=1115.089,-81.492,-47.555,179.692,4.866,148.918
C06863=1115.083,-81.242,-47.566,179.692,4.871,148.919
C06864=1115.079,-80.992,-47.576,179.692,4.876,148.921
C06865=1115.073,-80.743,-47.586,179.692,4.882,148.922
C06866=1115.068,-80.493,-47.596,179.692,4.887,148.923
C06867=1115.063,-80.243,-47.607,179.692,4.892,148.924
C06868=1115.057,-79.994,-47.617,179.692,4.897,148.925
C06869=1115.051,-79.744,-47.627,179.691,4.901,148.927
C06870=1115.046,-79.494,-47.638,179.691,4.907,148.928
C06871=1115.041,-79.244,-47.648,179.690,4.912,148.929
C06872=1115.036,-78.995,-47.657,179.690,4.917,148.930
C06873=1115.031,-78.745,-47.669,179.690,4.922,148.931
C06874=1115.026,-78.496,-47.679,179.690,4.927,148.932
C06875=1115.020,-78.246,-47.689,179.690,4.932,148.934
C06876=1115.015,-77.996,-47.700,179.690,4.938,148.935
C06877=1115.009,-77.747,-47.710,179.690,4.943,148.936
C06878=1115.004,-77.496,-47.721,179.690,4.949,148.937
C06879=1114.999,-77.247,-47.731,179.690,4.954,148.938
C06880=1114.993,-76.997,-47.741,179.690,4.959,148.939
C06881=1114.988,-76.747,-47.752,179.689,4.964,148.941
C06882=1114.983,-76.498,-47.762,179.689,4.969,148.942
C06883=1114.978,-76.248,-47.773,179.689,4.974,148.943
C06884=1114.972,-75.998,-47.783,179.689,4.979,148.944
C06885=1114.967,-75.749,-47.793,179.689,4.985,148.945
C06886=1114.962,-75.498,-47.804,179.689,4.990,148.946
C06887=1114.956,-75.249,-47.814,179.689,4.995,148.948
C06888=1114.951,-74.999,-47.825,179.689,5.000,148.949
C06889=1114.946,-74.750,-47.836,179.689,5.005,148.950
C06890=1114.941,-74.499,-47.846,179.689,5.011,148.951
C06891=1114.935,-74.250,-47.856,179.689,5.016,148.952
C06892=1114.930,-74.000,-47.867,179.689,5.021,148.953
C06893=1114.925,-73.751,-47.878,179.689,5.026,148.954
C06894=1114.921,-73.536,-47.887,179.689,5.030,148.955
C06895=1114.916,-73.321,-47.896,179.689,5.035,148.956
C06896=1114.911,-73.105,-47.905,179.689,5.040,148.957
C06897=1114.907,-72.891,-47.914,179.689,5.044,148.958
C06898=1114.902,-72.676,-47.923,179.689,5.049,148.959
C06899=1114.898,-72.460,-47.933,179.689,5.053,148.960
C06900=1114.893,-72.247,-47.942,179.689,5.057,148.961
C06901=1114.889,-72.031,-47.951,179.689,5.062,148.962
C06902=1114.883,-71.782,-47.961,179.689,5.067,148.963
C06903=1114.878,-71.531,-47.972,179.690,5.072,148.964
C06904=1114.873,-71.282,-47.983,179.689,5.077,148.965
C06905=1114.868,-71.032,-47.993,179.689,5.082,148.966
C06906=1114.862,-70.782,-48.004,179.689,5.088,148.968
C06907=1114.857,-70.533,-48.015,179.690,5.093,148.969
C06908=1114.852,-70.282,-48.026,179.690,5.098,148.970
C06909=1114.847,-70.034,-48.037,179.690,5.103,148.971
C06910=1114.842,-69.783,-48.047,179.690,5.108,148.972
C06911=1114.836,-69.534,-48.058,179.691,5.114,148.973
C06912=1114.831,-69.284,-48.069,179.691,5.119,148.974
C06913=1114.826,-69.035,-48.079,179.691,5.124,148.975
C06914=1114.820,-68.785,-48.091,179.691,5.129,148.976
C06915=1114.815,-68.535,-48.101,179.691,5.134,148.977
C06916=1114.810,-68.285,-48.112,179.692,5.140,148.978
C06917=1114.804,-68.036,-48.123,179.692,5.145,148.979
C06918=1114.799,-67.786,-48.133,179.692,5.150,148.980
C06919=1114.795,-67.536,-48.144,179.692,5.155,148.982
C06920=1114.788,-67.286,-48.155,179.693,5.161,148.982
C06921=1114.784,-67.037,-48.167,179.693,5.166,148.984
C06922=1114.778,-66.787,-48.177,179.693,5.170,148.985
C06923=1114.773,-66.537,-48.188,179.694,5.176,148.986
C06924=1114.767,-66.288,-48.199,179.694,5.181,148.987
C06925=1114.762,-66.038,-48.210,179.694,5.186,148.988
C06926=1114.757,-65.788,-48.221,179.694,5.191,148.989
C06927=1114.752,-65.539,-48.232,179.695,5.197,148.990
C06928=1114.747,-65.289,-48.243,179.695,5.202,148.991
C06929=1114.742,-65.039,-48.254,179.695,5.207,148.992
C06930=1114.736,-64.790,-48.265,179.696,5.212,148.993
C06931=1114.731,-64.539,-48.276,179.696,5.217,148.994
C06932=1114.725,-64.290,-48.287,179.696,5.222,148.995
C06933=1114.721,-64.041,-48.298,179.697,5.228,148.996
C06934=1114.716,-63.790,-48.309,179.697,5.233,148.997
C06935=1114.710,-63.541,-48.320,179.697,5.238,148.998
C06936=1114.705,-63.291,-48.331,179.698,5.243,148.999
C06937=1114.700,-63.041,-48.342,179.699,5.248,149.000
C06938=1114.695,-62.792,-48.353,179.699,5.253,149.001
C06939=1114.689,-62.542,-48.364,179.699,5.258,149.002
C06940=1114.684,-62.292,-48.376,179.700,5.264,149.003
C06941=1114.679,-62.043,-48.387,179.700,5.268,149.004
C06942=1114.673,-61.793,-48.399,179.701,5.274,149.005
C06943=1114.668,-61.543,-48.409,179.701,5.279,149.006
C06944=1114.663,-61.294,-48.420,179.702,5.284,149.007
C06945=1114.658,-61.044,-48.432,179.703,5.289,149.008
C06946=1114.653,-60.794,-48.443,179.703,5.294,149.009
C06947=1114.648,-60.544,-48.454,179.703,5.299,149.009
C06948=1114.642,-60.295,-48.465,179.704,5.304,149.010
C06949=1114.637,-60.045,-48.477,179.704,5.310,149.012
C06950=1114.633,-59.830,-48.486,179.704,5.313,149.012
C06951=1114.628,-59.615,-48.496,179.704,5.317,149.013
C06952=1114.623,-59.401,-48.506,179.704,5.321,149.014
C06953=1114.619,-59.186,-48.516,179.704,5.325,149.015
C06954=1114.614,-58.971,-48.525,179.704,5.330,149.016
C06955=1114.610,-58.756,-48.535,179.704,5.334,149.017
C06956=1114.606,-58.541,-48.545,179.704,5.338,149.018
C06957=1114.601,-58.326,-48.555,179.704,5.342,149.019
C06958=1114.596,-58.077,-48.566,179.703,5.346,149.020
C06959=1114.590,-57.826,-48.577,179.703,5.351,149.021
C06960=1114.586,-57.577,-48.588,179.703,5.356,149.022
C06961=1114.581,-57.327,-48.600,179.703,5.360,149.023
C06962=1114.575,-57.078,-48.611,179.703,5.365,149.024
C06963=1114.570,-56.828,-48.622,179.703,5.370,149.025
C06964=1114.565,-56.578,-48.634,179.702,5.374,149.026
C06965=1114.560,-56.329,-48.646,179.703,5.379,149.027
C06966=1114.555,-56.079,-48.657,179.702,5.383,149.028
C06967=1114.549,-55.829,-48.668,179.702,5.389,149.030
C06968=1114.544,-55.579,-48.680,179.702,5.393,149.030
C06969=1114.539,-55.330,-48.691,179.702,5.398,149.032
C06970=1114.534,-55.080,-48.703,179.702,5.402,149.033
C06971=1114.529,-54.830,-48.714,179.701,5.407,149.034
C06972=1114.523,-54.581,-48.725,179.701,5.412,149.035
C06973=1114.518,-54.331,-48.737,179.702,5.417,149.036
C06974=1114.513,-54.081,-48.749,179.701,5.421,149.037
C06975=1114.508,-53.832,-48.760,179.701,5.426,149.038
C06976=1114.503,-53.582,-48.772,179.701,5.431,149.039
C06977=1114.497,-53.333,-48.783,179.701,5.435,149.040
C06978=1114.492,-53.083,-48.795,179.701,5.440,149.041
C06979=1114.486,-52.833,-48.807,179.700,5.444,149.042
C06980=1114.482,-52.583,-48.818,179.700,5.449,149.043
C06981=1114.476,-52.333,-48.830,179.700,5.455,149.045
C06982=1114.472,-52.084,-48.841,179.700,5.458,149.045
C06983=1114.466,-51.835,-48.853,179.700,5.464,149.047
C06984=1114.461,-51.585,-48.864,179.699,5.468,149.048
C06985=1114.456,-51.335,-48.876,179.700,5.473,149.049
C06986=1114.450,-51.085,-48.888,179.700,5.478,149.050
C06987=1114.445,-50.835,-48.899,179.699,5.482,149.051
C06988=1114.440,-50.586,-48.911,179.699,5.487,149.052
C06989=1114.435,-50.337,-48.922,179.699,5.491,149.053
C06990=1114.429,-50.087,-48.934,179.699,5.496,149.054
C06991=1114.424,-49.837,-48.945,179.698,5.501,149.055
C06992=1114.419,-49.588,-48.957,179.698,5.505,149.056
C06993=1114.414,-49.338,-48.969,179.698,5.511,149.057
C06994=1114.409,-49.088,-48.981,179.698,5.516,149.059
C06995=1114.404,-48.838,-48.993,179.698,5.520,149.059
C06996=1114.398,-48.588,-49.004,179.698,5.525,149.061
C06997=1114.393,-48.339,-49.015,179.697,5.529,149.062
C06998=1114.388,-48.089,-49.027,179.697,5.534,149.063
C06999=1114.382,-47.840,-49.039,179.698,5.539,149.064
C07000=1114.378,-47.591,-49.051,179.697,5.543,149.065
C07001=1114.372,-47.341,-49.063,179.697,5.548,149.066
C07002=1114.367,-47.091,-49.075,179.697,5.552,149.067
C07003=1114.362,-46.841,-49.087,179.697,5.558,149.068
C07004=1114.357,-46.591,-49.098,179.697,5.563,149.069
C07005=1114.351,-46.341,-49.110,179.696,5.567,149.070
C07006=1114.346,-46.054,-49.124,179.696,5.572,149.072
C07007=1114.340,-45.768,-49.137,179.696,5.578,149.073
C07008=1114.334,-45.481,-49.151,179.696,5.584,149.074
C07009=1114.327,-45.193,-49.165,179.696,5.589,149.075
C07010=1114.323,-44.943,-49.176,179.695,5.593,149.076
C07011=1114.318,-44.694,-49.188,179.695,5.598,149.078
C07012=1114.312,-44.444,-49.200,179.695,5.603,149.079
C07013=1114.307,-44.194,-49.212,179.695,5.607,149.080
C07014=1114.302,-43.944,-49.224,179.695,5.612,149.081
C07015=1114.297,-43.695,-49.236,179.694,5.617,149.082
C07016=1114.291,-43.445,-49.248,179.694,5.621,149.083
C07017=1114.286,-43.195,-49.260,179.694,5.627,149.084
C07018=1114.282,-42.946,-49.272,179.694,5.631,149.085
C07019=1114.276,-42.696,-49.284,179.695,5.636,149.086
C07020=1114.271,-42.446,-49.296,179.696,5.642,149.087
C07021=1114.265,-42.198,-49.308,179.697,5.648,149.088
C07022=1114.260,-41.948,-49.319,179.697,5.652,149.089
C07023=1114.255,-41.698,-49.331,179.699,5.657,149.089
C07024=1114.250,-41.449,-49.344,179.700,5.663,149.090
C07025=1114.244,-41.199,-49.356,179.700,5.668,149.091
C07026=1114.239,-40.949,-49.367,179.701,5.673,149.092
C07027=1114.234,-40.699,-49.380,179.702,5.678,149.093
C07028=1114.229,-40.449,-49.392,179.703,5.683,149.094
C07029=1114.225,-40.200,-49.404,179.704,5.688,149.095
C07030=1114.216,-39.808,-49.424,179.705,5.696,149.096
C07031=1114.207,-39.416,-49.443,179.706,5.704,149.097
C07032=1114.199,-39.024,-49.461,179.708,5.712,149.099
C07033=1114.191,-38.632,-49.480,179.709,5.720,149.100
C07034=1114.186,-38.382,-49.493,179.709,5.724,149.101
C07035=1114.181,-38.132,-49.505,179.710,5.729,149.102
C07036=1114.175,-37.883,-49.517,179.711,5.733,149.103
C07037=1114.170,-37.633,-49.529,179.712,5.739,149.103
C07038=1114.166,-37.383,-49.542,179.713,5.743,149.104
C07039=1114.160,-37.133,-49.554,179.713,5.748,149.105
C07040=1114.155,-36.884,-49.567,179.713,5.753,149.106
C07041=1114.150,-36.634,-49.579,179.714,5.758,149.107
C07042=1114.144,-36.385,-49.591,179.715,5.762,149.108
C07043=1114.139,-36.135,-49.604,179.715,5.767,149.108
C07044=1114.134,-35.885,-49.616,179.716,5.771,149.109
C07045=1114.129,-35.636,-49.628,179.716,5.776,149.110
C07046=1114.123,-35.386,-49.640,179.717,5.780,149.111
C07047=1114.119,-35.136,-49.653,179.718,5.785,149.112
C07048=1114.114,-34.887,-49.666,179.718,5.790,149.113
C07049=1114.108,-34.637,-49.678,179.718,5.794,149.114
C07050=1114.103,-34.387,-49.690,179.718,5.799,149.115
C07051=1114.098,-34.138,-49.703,179.719,5.803,149.115
C07052=1114.093,-33.888,-49.715,179.720,5.808,149.116
C07053=1114.087,-33.639,-49.727,179.720,5.812,149.117
C07054=1114.083,-33.389,-49.740,179.720,5.816,149.118
C07055=1114.077,-33.139,-49.752,179.721,5.821,149.119
C07056=1114.072,-32.890,-49.765,179.721,5.826,149.120
C07057=1114.067,-32.640,-49.777,179.721,5.830,149.121
C07058=1114.063,-32.425,-49.787,179.721,5.833,149.121
C07059=1114.058,-32.211,-49.799,179.722,5.838,149.122
C07060=1114.054,-31.997,-49.809,179.722,5.842,149.123
C07061=1114.049,-31.781,-49.820,179.722,5.845,149.124
C07062=1114.046,-31.566,-49.831,179.722,5.849,149.124
C07063=1114.040,-31.351,-49.842,179.723,5.853,149.125
C07064=1114.036,-31.137,-49.852,179.722,5.857,149.126
C07065=1114.032,-30.923,-49.864,179.723,5.860,149.127
C07066=1114.026,-30.673,-49.876,179.723,5.864,149.128
C07067=1114.021,-30.423,-49.888,179.723,5.869,149.129
C07068=1114.017,-30.173,-49.901,179.723,5.873,149.129
C07069=1114.011,-29.924,-49.914,179.723,5.878,149.131
C07070=1114.006,-29.675,-49.926,179.723,5.882,149.132
C07071=1114.001,-29.425,-49.938,179.723,5.887,149.132
C07072=1113.995,-29.175,-49.951,179.723,5.890,149.133
C07073=1113.991,-28.925,-49.964,179.723,5.894,149.134
C07074=1113.985,-28.676,-49.977,179.723,5.900,149.135
C07075=1113.980,-28.426,-49.990,179.723,5.903,149.136
C07076=1113.975,-28.177,-50.002,179.723,5.907,149.137
C07077=1113.971,-27.927,-50.015,179.722,5.912,149.138
C07078=1113.965,-27.677,-50.027,179.722,5.916,149.139
C07079=1113.959,-27.427,-50.040,179.722,5.920,149.140
C07080=1113.954,-27.178,-50.053,179.722,5.925,149.141
C07081=1113.950,-26.928,-50.066,179.722,5.929,149.142
C07082=1113.945,-26.679,-50.078,179.722,5.934,149.143
C07083=1113.939,-26.430,-50.091,179.721,5.938,149.144
C07084=1113.934,-26.180,-50.104,179.721,5.942,149.145
C07085=1113.929,-25.930,-50.117,179.720,5.946,149.146
C07086=1113.924,-25.681,-50.130,179.721,5.951,149.147
C07087=1113.919,-25.431,-50.142,179.721,5.956,149.148
C07088=1113.914,-25.181,-50.155,179.722,5.961,149.149
C07089=1113.908,-24.931,-50.168,179.722,5.966,149.150
C07090=1113.903,-24.682,-50.180,179.722,5.970,149.151
C07091=1113.898,-24.432,-50.193,179.723,5.975,149.152
C07092=1113.893,-24.182,-50.206,179.723,5.980,149.153
C07093=1113.888,-23.933,-50.219,179.724,5.985,149.154
C07094=1113.882,-23.683,-50.232,179.724,5.989,149.155
C07095=1113.878,-23.433,-50.245,179.724,5.994,149.156
C07096=1113.873,-23.184,-50.257,179.725,5.999,149.157
C07097=1113.867,-22.934,-50.271,179.725,6.004,149.157
C07098=1113.862,-22.685,-50.283,179.726,6.008,149.158
C07099=1113.857,-22.435,-50.296,179.726,6.013,149.159
C07100=1113.851,-22.185,-50.309,179.727,6.018,149.160
C07101=1113.846,-21.936,-50.322,179.727,6.022,149.161
C07102=1113.842,-21.686,-50.335,179.728,6.027,149.162
C07103=1113.836,-21.436,-50.348,179.728,6.032,149.163
C07104=1113.831,-21.188,-50.361,179.729,6.036,149.164
C07105=1113.827,-20.938,-50.374,179.730,6.041,149.164
C07106=1113.821,-20.688,-50.388,179.730,6.046,149.165
C07107=1113.816,-20.438,-50.400,179.731,6.050,149.166
C07108=1113.811,-20.189,-50.413,179.731,6.055,149.167
C07109=1113.805,-19.939,-50.426,179.732,6.060,149.168
C07110=1113.801,-19.689,-50.439,179.732,6.065,149.169
C07111=1113.796,-19.440,-50.452,179.733,6.069,149.170
C07112=1113.790,-19.191,-50.466,179.733,6.074,149.171
C07113=1113.785,-18.941,-50.479,179.734,6.079,149.172
C07114=1113.781,-18.726,-50.490,179.735,6.083,149.172
C07115=1113.776,-18.512,-50.501,179.735,6.087,149.173
C07116=1113.772,-18.297,-50.512,179.735,6.091,149.174
C07117=1113.768,-18.082,-50.524,179.736,6.095,149.175
C07118=1113.763,-17.868,-50.535,179.736,6.099,149.175
C07119=1113.758,-17.653,-50.546,179.737,6.103,149.176
C07120=1113.755,-17.438,-50.557,179.737,6.107,149.177
C07121=1113.750,-17.224,-50.569,179.738,6.111,149.177
C07122=1113.744,-16.974,-50.582,179.739,6.116,149.178
C07123=1113.740,-16.725,-50.596,179.739,6.121,149.179
C07124=1113.734,-16.475,-50.609,179.740,6.125,149.180
C07125=1113.729,-16.225,-50.622,179.740,6.130,149.181
C07126=1113.725,-15.976,-50.635,179.741,6.134,149.182
C07127=1113.719,-15.727,-50.648,179.741,6.138,149.183
C07128=1113.714,-15.477,-50.661,179.741,6.143,149.183
C07129=1113.708,-15.227,-50.675,179.742,6.148,149.184
C07130=1113.704,-14.978,-50.688,179.743,6.152,149.185
C07131=1113.698,-14.728,-50.701,179.743,6.157,149.186
C07132=1113.694,-14.478,-50.714,179.744,6.162,149.187
C07133=1113.688,-14.229,-50.728,179.744,6.166,149.188
C07134=1113.684,-13.979,-50.741,179.745,6.171,149.189
C07135=1113.678,-13.730,-50.755,179.746,6.175,149.189
C07136=1113.674,-13.480,-50.768,179.746,6.180,149.190
C07137=1113.668,-13.230,-50.781,179.747,6.185,149.191
C07138=1113.663,-12.980,-50.796,179.747,6.190,149.192
C07139=1113.658,-12.731,-50.808,179.748,6.194,149.193
C07140=1113.653,-12.481,-50.822,179.749,6.199,149.194
C07141=1113.648,-12.232,-50.835,179.749,6.203,149.194
C07142=1113.642,-11.982,-50.849,179.749,6.207,149.195
C07143=1113.638,-11.733,-50.862,179.750,6.212,149.196
C07144=1113.632,-11.483,-50.876,179.751,6.216,149.197
C07145=1113.627,-11.234,-50.889,179.751,6.221,149.198
C07146=1113.622,-10.984,-50.902,179.752,6.226,149.199
C07147=1113.617,-10.735,-50.916,179.753,6.230,149.199
C07148=1113.612,-10.485,-50.929,179.753,6.235,149.200
C07149=1113.607,-10.235,-50.944,179.754,6.240,149.201
C07150=1113.601,-9.985,-50.957,179.754,6.244,149.202
C07151=1113.597,-9.736,-50.970,179.755,6.249,149.203
C07152=1113.591,-9.486,-50.984,179.756,6.253,149.204
C07153=1113.587,-9.237,-50.997,179.756,6.258,149.204
C07154=1113.581,-8.987,-51.010,179.756,6.262,149.205
C07155=1113.576,-8.738,-51.025,179.757,6.266,149.206
C07156=1113.571,-8.489,-51.038,179.758,6.271,149.207
C07157=1113.566,-8.239,-51.052,179.758,6.276,149.208
C07158=1113.561,-7.989,-51.066,179.759,6.280,149.208
C07159=1113.556,-7.740,-51.079,179.760,6.285,149.209
C07160=1113.551,-7.490,-51.093,179.760,6.290,149.210
C07161=1113.546,-7.241,-51.107,179.761,6.294,149.211
C07162=1113.540,-6.991,-51.120,179.762,6.299,149.212
C07163=1113.536,-6.741,-51.134,179.762,6.303,149.213
C07164=1113.530,-6.491,-51.147,179.762,6.307,149.214
C07165=1113.525,-6.242,-51.161,179.763,6.312,149.214
C07166=1113.520,-5.993,-51.175,179.764,6.316,149.215
C07167=1113.515,-5.743,-51.188,179.764,6.321,149.216
C07168=1113.510,-5.493,-51.203,179.765,6.326,149.217
C07169=1113.505,-5.244,-51.217,179.766,6.330,149.218
C07170=1113.501,-5.029,-51.228,179.766,6.334,149.218
C07171=1113.496,-4.815,-51.240,179.766,6.338,149.219
C07172=1113.492,-4.600,-51.252,179.767,6.342,149.220
C07173=1113.487,-4.386,-51.264,179.767,6.345,149.221
C07174=1113.483,-4.170,-51.276,179.768,6.350,149.221
C07175=1113.479,-3.956,-51.288,179.769,6.353,149.222
C07176=1113.474,-3.743,-51.300,179.769,6.357,149.223
C07177=1113.470,-3.527,-51.311,179.770,6.362,149.223
C07178=1113.465,-3.278,-51.326,179.771,6.366,149.224
C07179=1113.460,-3.029,-51.340,179.771,6.371,149.225
C07180=1113.455,-2.779,-51.353,179.771,6.375,149.226
C07181=1113.450,-2.529,-51.367,179.771,6.379,149.227
C07182=1113.445,-2.280,-51.381,179.772,6.384,149.227
C07183=1113.440,-2.030,-51.395,179.773,6.388,149.228
C07184=1113.435,-1.780,-51.409,179.774,6.393,149.229
C07185=1113.429,-1.531,-51.422,179.775,6.397,149.230
C07186=1113.424,-1.281,-51.437,179.775,6.402,149.231
C07187=1113.420,-1.032,-51.450,179.776,6.407,149.232
C07188=1113.414,-0.783,-51.464,179.776,6.412,149.233
C07189=1113.409,-0.533,-51.479,179.777,6.415,149.233
C07190=1113.404,-0.283,-51.493,179.777,6.420,149.234
C07191=1113.399,-0.034,-51.507,179.778,6.424,149.235
C07192=1113.394,0.215,-51.521,179.779,6.429,149.236
C07193=1113.388,0.466,-51.535,179.779,6.434,149.237
C07194=1113.383,0.716,-51.549,179.780,6.438,149.237
C07195=1113.379,0.965,-51.563,179.780,6.443,149.238
C07196=1113.373,1.214,-51.577,179.781,6.447,149.239
C07197=1113.369,1.464,-51.591,179.782,6.452,149.240
C07198=1113.364,1.713,-51.605,179.782,6.457,149.241
C07199=1113.359,1.963,-51.619,179.782,6.461,149.242
C07200=1113.353,2.212,-51.633,179.783,6.465,149.242
C07201=1113.348,2.462,-51.648,179.784,6.470,149.243
C07202=1113.343,2.711,-51.662,179.784,6.474,149.244
C07203=1113.338,2.961,-51.676,179.785,6.479,149.245
C07204=1113.333,3.210,-51.690,179.786,6.483,149.246
C07205=1113.328,3.460,-51.704,179.786,6.488,149.246
C07206=1113.323,3.710,-51.719,179.787,6.493,149.247
C07207=1113.318,3.959,-51.733,179.787,6.498,149.248
C07208=1113.313,4.209,-51.747,179.788,6.502,149.249
C07209=1113.307,4.458,-51.761,179.789,6.507,149.250
C07210=1113.303,4.708,-51.775,179.789,6.511,149.251
C07211=1113.298,4.957,-51.790,179.789,6.515,149.252
C07212=1113.293,5.207,-51.804,179.790,6.520,149.252
C07213=1113.288,5.456,-51.819,179.791,6.524,149.253
C07214=1113.283,5.706,-51.833,179.791,6.529,149.254
C07215=1113.277,5.955,-51.847,179.792,6.534,149.255
C07216=1113.273,6.205,-51.861,179.793,6.538,149.256
C07217=1113.268,6.454,-51.876,179.793,6.543,149.257
C07218=1113.263,6.704,-51.890,179.794,6.547,149.257
C07219=1113.257,6.954,-51.905,179.795,6.552,149.258
C07220=1113.252,7.203,-51.920,179.795,6.557,149.259
C07221=1113.247,7.453,-51.934,179.796,6.562,149.260
C07222=1113.242,7.702,-51.948,179.796,6.566,149.261
C07223=1113.237,7.952,-51.962,179.796,6.570,149.262
C07224=1113.232,8.201,-51.976,179.797,6.575,149.262
C07225=1113.227,8.451,-51.991,179.798,6.579,149.263
C07226=1113.223,8.666,-52.003,179.798,6.584,149.264
C07227=1113.218,8.880,-52.016,179.799,6.588,149.265
C07228=1113.214,9.095,-52.028,179.799,6.591,149.266
C07229=1113.209,9.309,-52.040,179.800,6.596,149.266
C07230=1113.205,9.524,-52.053,179.800,6.599,149.267
C07231=1113.201,9.738,-52.066,179.801,6.603,149.268
C07232=1113.197,9.951,-52.078,179.802,6.607,149.268
C07233=1113.192,10.166,-52.091,179.801,6.611,149.269
C07234=1113.187,10.416,-52.106,179.802,6.616,149.270
C07235=1113.182,10.666,-52.120,179.803,6.620,149.271
C07236=1113.177,10.916,-52.134,179.804,6.625,149.272
C07237=1113.172,11.165,-52.150,179.804,6.630,149.273
C07238=1113.166,11.414,-52.164,179.804,6.633,149.273
C07239=1113.161,11.664,-52.178,179.805,6.638,149.274
C07240=1113.157,11.913,-52.193,179.806,6.642,149.275
C07241=1113.152,12.162,-52.207,179.806,6.647,149.276
C07242=1113.146,12.412,-52.222,179.807,6.652,149.277
C07243=1113.142,12.662,-52.237,179.808,6.656,149.277
C07244=1113.137,12.911,-52.251,179.808,6.661,149.278
C07245=1113.132,13.160,-52.266,179.809,6.666,149.279
C07246=1113.126,13.410,-52.281,179.809,6.669,149.280
C07247=1113.121,13.660,-52.295,179.810,6.674,149.281
C07248=1113.117,13.909,-52.310,179.810,6.679,149.282
C07249=1113.112,14.159,-52.325,179.811,6.683,149.282
C07250=1113.106,14.408,-52.340,179.812,6.688,149.283
C07251=1113.101,14.658,-52.355,179.813,6.692,149.284
C07252=1113.097,14.907,-52.370,179.814,6.697,149.285
C07253=1113.092,15.157,-52.384,179.814,6.701,149.286
C07254=1113.086,15.406,-52.399,179.814,6.705,149.286
C07255=1113.081,15.656,-52.414,179.815,6.710,149.287
C07256=1113.077,15.905,-52.429,179.816,6.714,149.288
C07257=1113.071,16.155,-52.444,179.816,6.719,149.289
C07258=1113.066,16.404,-52.459,179.817,6.723,149.290
C07259=1113.061,16.654,-52.473,179.818,6.728,149.290
C07260=1113.056,16.903,-52.488,179.819,6.732,149.291
C07261=1113.051,17.153,-52.503,179.819,6.736,149.292
C07262=1113.046,17.402,-52.518,179.820,6.741,149.293
C07263=1113.041,17.652,-52.533,179.820,6.745,149.293
C07264=1113.036,17.901,-52.548,179.821,6.750,149.294
C07265=1113.031,18.151,-52.562,179.822,6.754,149.295
C07266=1113.026,18.400,-52.577,179.823,6.759,149.296
C07267=1113.021,18.649,-52.592,179.824,6.763,149.297
C07268=1113.015,18.899,-52.607,179.824,6.767,149.297
C07269=1113.011,19.148,-52.622,179.825,6.772,149.298
C07270=1113.006,19.399,-52.637,179.825,6.776,149.299
C07271=1113.001,19.648,-52.653,179.826,6.781,149.300
C07272=1112.996,19.897,-52.668,179.827,6.785,149.301
C07273=1112.991,20.147,-52.682,179.828,6.790,149.301
C07274=1112.986,20.397,-52.697,179.829,6.794,149.302
C07275=1112.981,20.646,-52.713,179.829,6.798,149.303
C07276=1112.976,20.896,-52.727,179.830,6.802,149.303
C07277=1112.971,21.145,-52.742,179.831,6.807,149.304
C07278=1112.966,21.394,-52.758,179.832,6.811,149.305
C07279=1112.961,21.644,-52.772,179.832,6.816,149.306
C07280=1112.955,21.893,-52.788,179.833,6.820,149.306
C07281=1112.951,22.143,-52.803,179.834,6.824,149.307
C07282=1112.946,22.357,-52.816,179.835,6.828,149.308
C07283=1112.942,22.572,-52.829,179.835,6.832,149.308
C07284=1112.938,22.786,-52.842,179.836,6.835,149.309
C07285=1112.934,23.001,-52.856,179.837,6.839,149.310
C07286=1112.929,23.214,-52.868,179.837,6.843,149.310
C07287=1112.925,23.429,-52.881,179.837,6.846,149.311
C07288=1112.920,23.644,-52.894,179.838,6.851,149.312
C07289=1112.917,23.858,-52.907,179.839,6.854,149.312
C07290=1112.911,24.107,-52.923,179.840,6.859,149.313
C07291=1112.907,24.356,-52.938,179.841,6.863,149.314
C07292=1112.901,24.606,-52.953,179.841,6.866,149.314
C07293=1112.896,24.856,-52.968,179.842,6.871,149.315
C07294=1112.892,25.105,-52.984,179.843,6.875,149.316
C07295=1112.886,25.355,-52.999,179.844,6.880,149.317
C07296=1112.882,25.604,-53.014,179.845,6.884,149.317
C07297=1112.876,25.853,-53.030,179.845,6.888,149.318
C07298=1112.871,26.103,-53.044,179.846,6.892,149.319
C07299=1112.866,26.353,-53.060,179.847,6.897,149.319
C07300=1112.861,26.603,-53.076,179.848,6.901,149.320
C07301=1112.856,26.852,-53.091,179.849,6.906,149.321
C07302=1112.851,27.101,-53.106,179.850,6.910,149.322
C07303=1112.846,27.350,-53.121,179.850,6.913,149.322
C07304=1112.842,27.600,-53.137,179.851,6.918,149.323
C07305=1112.836,27.850,-53.153,179.852,6.922,149.324
C07306=1112.832,28.099,-53.168,179.853,6.927,149.324
C07307=1112.826,28.348,-53.183,179.854,6.931,149.325
C07308=1112.821,28.598,-53.199,179.855,6.935,149.326
C07309=1112.817,28.847,-53.214,179.855,6.939,149.327
C07310=1112.811,29.097,-53.230,179.856,6.944,149.327
C07311=1112.806,29.346,-53.246,179.857,6.948,149.328
C07312=1112.802,29.596,-53.261,179.858,6.952,149.329
C07313=1112.796,29.845,-53.277,179.859,6.957,149.329
C07314=1112.791,30.095,-53.292,179.860,6.961,149.330
C07315=1112.786,30.344,-53.307,179.860,6.965,149.331
C07316=1112.782,30.594,-53.323,179.861,6.969,149.331
C07317=1112.776,30.843,-53.339,179.862,6.973,149.332
C07318=1112.771,31.093,-53.354,179.864,6.978,149.333
C07319=1112.766,31.342,-53.369,179.865,6.982,149.333
C07320=1112.761,31.592,-53.385,179.865,6.986,149.334
